Universal Robots PolyScope program: azat-test.urp

Program azat-test (installation=default directory=/programs createdIn=5.11.9.1010452 lastSavedIn=5.11.9.1010452 robotSerialNumber=20225200364)
Calibrated DH parameters: a=[0.00002, -0.569483, -0.54992, -0.00001, -0.000036, 0]; d=[0.180894, -146.691669, 192.918669, -46.053088, 0.119778, 0.115602]; alpha=[1.571425, -0.001534, 0.003359, 1.568739, -1.571477, 0]; deltaTheta=[0, 0.376258, -0.101074, -0.275185, -0.000002, 0]
Robot Program (runOnlyOnce=false)
  Script file /programs/usbdisk/Test.script
    | def Machining2():
    |   # Default parameters:
    |   global speed_ms = 0.3
    |   global speed_rads = 0.75
    |   global accel_mss = 3
    |   global accel_radss = 1.2
    |   global blend_radius_m = 0.001
    | 
    |   # Add subprograms here
    |   # Start of main program
    |   # Program generated by RoboDK v5.6.5 for UR10e on 11/10/2023 19:05:33
    |   # Using nominal kinematics.
    |   blend_radius_m = 0.001
    |   speed_ms = 1.000
    |   # set_reference(p[0.335000, -0.154000, 0.000000, 0.000000, 0.000000, 0.000000])
    |   set_tcp(p[0.000000, 0.000000, 0.252000, 0.000000, 0.000000, 0.000000])
    |   # Show Tool
    |   movej([0.093203, -1.219144, -2.564771, -0.928474, 1.570796, 1.664000],accel_radss,speed_rads,0,blend_radius_m)
    |   movel([0.093203, -1.219144, -2.564771, -0.928474, 1.570796, 1.664000],accel_mss,speed_ms,0,blend_radius_m)
    |   # Splitting Linear movement in 32 (instruction 7: MoveL 3)
    |   movel([0.093203, -1.220829, -2.565913, -0.925646, 1.570796, 1.664000],accel_mss,speed_ms,0,blend_radius_m)
    |   movel([0.093203, -1.222524, -2.567053, -0.922812, 1.570796, 1.664000],accel_mss,speed_ms,0,blend_radius_m)
    |   movel([0.093203, -1.224229, -2.568190, -0.919970, 1.570796, 1.664000],accel_mss,speed_ms,0,blend_radius_m)
    |   movel([0.093203, -1.225943, -2.569325, -0.917122, 1.570796, 1.664000],accel_mss,speed_ms,0,blend_radius_m)
    |   movel([0.093203, -1.227666, -2.570456, -0.914267, 1.570796, 1.664000],accel_mss,speed_ms,0,blend_radius_m)
    |   movel([0.093203, -1.229398, -2.571586, -0.911405, 1.570796, 1.664000],accel_mss,speed_ms,0,blend_radius_m)
    |   movel([0.093203, -1.231141, -2.572712, -0.908536, 1.570796, 1.664000],accel_mss,speed_ms,0,blend_radius_m)
    |   movel([0.093203, -1.232892, -2.573836, -0.905661, 1.570796, 1.664000],accel_mss,speed_ms,0,blend_radius_m)
    |   movel([0.093203, -1.234653, -2.574957, -0.902778, 1.570796, 1.664000],accel_mss,speed_ms,0,blend_radius_m)
    |   movel([0.093203, -1.236424, -2.576076, -0.899889, 1.570796, 1.664000],accel_mss,speed_ms,0,blend_radius_m)
    |   movel([0.093203, -1.238204, -2.577191, -0.896993, 1.570796, 1.664000],accel_mss,speed_ms,0,blend_radius_m)
    |   movel([0.093203, -1.239994, -2.578304, -0.894090, 1.570796, 1.664000],accel_mss,speed_ms,0,blend_radius_m)
    |   movel([0.093203, -1.241794, -2.579415, -0.891180, 1.570796, 1.664000],accel_mss,speed_ms,0,blend_radius_m)
    |   movel([0.093203, -1.243603, -2.580522, -0.888264, 1.570796, 1.664000],accel_mss,speed_ms,0,blend_radius_m)
    |   movel([0.093203, -1.245422, -2.581627, -0.885340, 1.570796, 1.664000],accel_mss,speed_ms,0,blend_radius_m)
    |   movel([0.093203, -1.247251, -2.582729, -0.882409, 1.570796, 1.664000],accel_mss,speed_ms,0,blend_radius_m)
    |   movel([0.093203, -1.249090, -2.583828, -0.879472, 1.570796, 1.664000],accel_mss,speed_ms,0,blend_radius_m)
    |   movel([0.093203, -1.250938, -2.584924, -0.876527, 1.570796, 1.664000],accel_mss,speed_ms,0,blend_radius_m)
    |   movel([0.093203, -1.252796, -2.586018, -0.873575, 1.570796, 1.664000],accel_mss,speed_ms,0,blend_radius_m)
    |   movel([0.093203, -1.254664, -2.587108, -0.870617, 1.570796, 1.664000],accel_mss,speed_ms,0,blend_radius_m)
    |   movel([0.093203, -1.256542, -2.588196, -0.867651, 1.570796, 1.664000],accel_mss,speed_ms,0,blend_radius_m)
    |   movel([0.093203, -1.258430, -2.589281, -0.864678, 1.570796, 1.664000],accel_mss,speed_ms,0,blend_radius_m)
    |   movel([0.093203, -1.260327, -2.590363, -0.861699, 1.570796, 1.664000],accel_mss,speed_ms,0,blend_radius_m)
    |   movel([0.093203, -1.262235, -2.591442, -0.858712, 1.570796, 1.664000],accel_mss,speed_ms,0,blend_radius_m)
    |   movel([0.093203, -1.264153, -2.592518, -0.855718, 1.570796, 1.664000],accel_mss,speed_ms,0,blend_radius_m)
    |   movel([0.093203, -1.266080, -2.593592, -0.852717, 1.570796, 1.664000],accel_mss,speed_ms,0,blend_radius_m)
    |   movel([0.093203, -1.268018, -2.594662, -0.849709, 1.570796, 1.664000],accel_mss,speed_ms,0,blend_radius_m)
    |   movel([0.093203, -1.269966, -2.595730, -0.846694, 1.570796, 1.664000],accel_mss,speed_ms,0,blend_radius_m)
    |   movel([0.093203, -1.271924, -2.596794, -0.843671, 1.570796, 1.664000],accel_mss,speed_ms,0,blend_radius_m)
    |   movel([0.093203, -1.273891, -2.597855, -0.840642, 1.570796, 1.664000],accel_mss,speed_ms,0,blend_radius_m)
    |   movel([0.093203, -1.275870, -2.598914, -0.837605, 1.570796, 1.664000],accel_mss,speed_ms,0,blend_radius_m)
    |   movel([0.093203, -1.277858, -2.599969, -0.834562, 1.570796, 1.664000],accel_mss,speed_ms,0,blend_radius_m)
    |   movel([0.093203, -1.277858, -2.599969, -0.834562, 1.570796, 1.664000],accel_mss,speed_ms,0,blend_radius_m)
    |   speed_ms = 1.000
    |   movel([0.093203, -1.277858, -2.599969, -0.834562, 1.570796, 1.664000],accel_mss,speed_ms,0,blend_radius_m)
    |   # Splitting Linear movement in 14 (instruction 11: MoveL 6)
    |   movel([0.093203, -1.279685, -2.600932, -0.831772, 1.570796, 1.664000],accel_mss,speed_ms,0,blend_radius_m)
    |   movel([0.093203, -1.281520, -2.601892, -0.828977, 1.570796, 1.664000],accel_mss,speed_ms,0,blend_radius_m)
    |   movel([0.093203, -1.283364, -2.602849, -0.826176, 1.570796, 1.664000],accel_mss,speed_ms,0,blend_radius_m)
    |   movel([0.093203, -1.285216, -2.603804, -0.823369, 1.570796, 1.664000],accel_mss,speed_ms,0,blend_radius_m)
    |   movel([0.093203, -1.287077, -2.604756, -0.820556, 1.570796, 1.664000],accel_mss,speed_ms,0,blend_radius_m)
    |   movel([0.093203, -1.288947, -2.605705, -0.817737, 1.570796, 1.664000],accel_mss,speed_ms,0,blend_radius_m)
    |   movel([0.093203, -1.290825, -2.606652, -0.814911, 1.570796, 1.664000],accel_mss,speed_ms,0,blend_radius_m)
    |   movel([0.093203, -1.292712, -2.607597, -0.812080, 1.570796, 1.664000],accel_mss,speed_ms,0,blend_radius_m)
    |   movel([0.093203, -1.294608, -2.608538, -0.809243, 1.570796, 1.664000],accel_mss,speed_ms,0,blend_radius_m)
    |   movel([0.093203, -1.296512, -2.609477, -0.806399, 1.570796, 1.664000],accel_mss,speed_ms,0,blend_radius_m)
    |   movel([0.093203, -1.298425, -2.610414, -0.803550, 1.570796, 1.664000],accel_mss,speed_ms,0,blend_radius_m)
    |   movel([0.093203, -1.300347, -2.611348, -0.800694, 1.570796, 1.664000],accel_mss,speed_ms,0,blend_radius_m)
    |   movel([0.093203, -1.302278, -2.612279, -0.797833, 1.570796, 1.664000],accel_mss,speed_ms,0,blend_radius_m)
    |   movel([0.093203, -1.304217, -2.613207, -0.794965, 1.570796, 1.664000],accel_mss,speed_ms,0,blend_radius_m)
    |   speed_ms = 0.003
    |   # Splitting Linear movement in 6 (instruction 13: MoveL 7)
    |   movel([0.093203, -1.305921, -2.614017, -0.792451, 1.570796, 1.664000],accel_mss,speed_ms,0,blend_radius_m)
    |   movel([0.093203, -1.307632, -2.614825, -0.789932, 1.570796, 1.664000],accel_mss,speed_ms,0,blend_radius_m)
    |   movel([0.093203, -1.309349, -2.615632, -0.787408, 1.570796, 1.664000],accel_mss,speed_ms,0,blend_radius_m)
    |   movel([0.093203, -1.311073, -2.616435, -0.784880, 1.570796, 1.664000],accel_mss,speed_ms,0,blend_radius_m)
    |   movel([0.093203, -1.312805, -2.617237, -0.782347, 1.570796, 1.664000],accel_mss,speed_ms,0,blend_radius_m)
    |   movel([0.093203, -1.314542, -2.618037, -0.779810, 1.570796, 1.664000],accel_mss,speed_ms,0,blend_radius_m)
    |   speed_ms = 0.007
    |   # Splitting Linear movement in 4 (instruction 15: MoveC 8)
    |   movel([0.093414, -1.312771, -2.619122, -0.780496, 1.570796, 1.664211],accel_mss,speed_ms,0,blend_radius_m)
    |   movel([0.093626, -1.310995, -2.620205, -0.781189, 1.570796, 1.664423],accel_mss,speed_ms,0,blend_radius_m)
    |   movel([0.093839, -1.309214, -2.621287, -0.781888, 1.570796, 1.664635],accel_mss,speed_ms,0,blend_radius_m)
    |   movel([0.094053, -1.307428, -2.622368, -0.782593, 1.570796, 1.664849],accel_mss,speed_ms,0,blend_radius_m)
    |   movel([0.094549, -1.306453, -2.622956, -0.782979, 1.570796, 1.665345],accel_mss,speed_ms,0,blend_radius_m)
    |   movel([0.095474, -1.305833, -2.623330, -0.783226, 1.570796, 1.666271],accel_mss,speed_ms,0,blend_radius_m)
    |   # Splitting Linear movement in 4 (instruction 18: MoveC 11)
    |   movel([0.097666, -1.305097, -2.623773, -0.783519, 1.570796, 1.668462],accel_mss,speed_ms,0,blend_radius_m)
    |   movel([0.099859, -1.304363, -2.624214, -0.783812, 1.570796, 1.670655],accel_mss,speed_ms,0,blend_radius_m)
    |   movel([0.102053, -1.303632, -2.624652, -0.784105, 1.570796, 1.672850],accel_mss,speed_ms,0,blend_radius_m)
    |   movel([0.104249, -1.302904, -2.625088, -0.784397, 1.570796, 1.675046],accel_mss,speed_ms,0,blend_radius_m)
    |   # Splitting Linear movement in 4 (instruction 19: MoveC 12)
    |   movel([0.106367, -1.302217, -2.625498, -0.784673, 1.570796, 1.677163],accel_mss,speed_ms,0,blend_radius_m)
    |   movel([0.108485, -1.301533, -2.625907, -0.784949, 1.570796, 1.679281],accel_mss,speed_ms,0,blend_radius_m)
    |   movel([0.110605, -1.300852, -2.626313, -0.785224, 1.570796, 1.681401],accel_mss,speed_ms,0,blend_radius_m)
    |   movel([0.112726, -1.300173, -2.626717, -0.785499, 1.570796, 1.683522],accel_mss,speed_ms,0,blend_radius_m)
    |   movel([0.114487, -1.299907, -2.626875, -0.785607, 1.570796, 1.685284],accel_mss,speed_ms,0,blend_radius_m)
    |   movel([0.114805, -1.300192, -2.626705, -0.785491, 1.570796, 1.685601],accel_mss,speed_ms,0,blend_radius_m)
    |   movel([0.114810, -1.301339, -2.626023, -0.785027, 1.570796, 1.685607],accel_mss,speed_ms,0,blend_radius_m)
    |   movel([0.114595, -1.303476, -2.624746, -0.784167, 1.570796, 1.685391],accel_mss,speed_ms,0,blend_radius_m)
    |   movel([0.113935, -1.308261, -2.621865, -0.782263, 1.570796, 1.684731],accel_mss,speed_ms,0,blend_radius_m)
    |   movel([0.113353, -1.312385, -2.619358, -0.780647, 1.570796, 1.684149],accel_mss,speed_ms,0,blend_radius_m)
    |   movel([0.112775, -1.316484, -2.616843, -0.779061, 1.570796, 1.683572],accel_mss,speed_ms,0,blend_radius_m)
    |   movel([0.107814, -1.318044, -2.615881, -0.778464, 1.570796, 1.678611],accel_mss,speed_ms,0,blend_radius_m)
    |   movel([0.102861, -1.319618, -2.614906, -0.777865, 1.570796, 1.673657],accel_mss,speed_ms,0,blend_radius_m)
    |   movel([0.097870, -1.321202, -2.613922, -0.777265, 1.570796, 1.668666],accel_mss,speed_ms,0,blend_radius_m)
    |   movel([0.094990, -1.322063, -2.613386, -0.776941, 1.570796, 1.665786],accel_mss,speed_ms,0,blend_radius_m)
    |   movel([0.093115, -1.322559, -2.613076, -0.776754, 1.570796, 1.663912],accel_mss,speed_ms,0,blend_radius_m)
    |   movel([0.092693, -1.322465, -2.613135, -0.776789, 1.570796, 1.663490],accel_mss,speed_ms,0,blend_radius_m)
    |   movel([0.092441, -1.321460, -2.613761, -0.777168, 1.570796, 1.663237],accel_mss,speed_ms,0,blend_radius_m)
    |   # Splitting Linear movement in 4 (instruction 34: MoveC 27)
    |   movel([0.092630, -1.319737, -2.614832, -0.777820, 1.570796, 1.663427],accel_mss,speed_ms,0,blend_radius_m)
    |   movel([0.092821, -1.318010, -2.615902, -0.778477, 1.570796, 1.663617],accel_mss,speed_ms,0,blend_radius_m)
    |   movel([0.093012, -1.316279, -2.616970, -0.779140, 1.570796, 1.663808],accel_mss,speed_ms,0,blend_radius_m)
    |   movel([0.093203, -1.314542, -2.618037, -0.779810, 1.570796, 1.664000],accel_mss,speed_ms,0,blend_radius_m)
    |   speed_ms = 0.003
    |   movel([0.093203, -1.318038, -2.619630, -0.774720, 1.570796, 1.664000],accel_mss,speed_ms,0,blend_radius_m)
    |   speed_ms = 0.007
    |   # Splitting Linear movement in 4 (instruction 38: MoveC 29)
    |   movel([0.093414, -1.316271, -2.620718, -0.775400, 1.570796, 1.664211],accel_mss,speed_ms,0,blend_radius_m)
    |   movel([0.093626, -1.314500, -2.621804, -0.776085, 1.570796, 1.664423],accel_mss,speed_ms,0,blend_radius_m)
    |   movel([0.093839, -1.312723, -2.622889, -0.776777, 1.570796, 1.664635],accel_mss,speed_ms,0,blend_radius_m)
    |   movel([0.094053, -1.310941, -2.623973, -0.777474, 1.570796, 1.664849],accel_mss,speed_ms,0,blend_radius_m)
    |   movel([0.094549, -1.309969, -2.624563, -0.777857, 1.570796, 1.665345],accel_mss,speed_ms,0,blend_radius_m)
    |   movel([0.095474, -1.309350, -2.624938, -0.778101, 1.570796, 1.666271],accel_mss,speed_ms,0,blend_radius_m)
    |   # Splitting Linear movement in 4 (instruction 41: MoveC 32)
    |   movel([0.097666, -1.308615, -2.625382, -0.778391, 1.570796, 1.668462],accel_mss,speed_ms,0,blend_radius_m)
    |   movel([0.099859, -1.307884, -2.625824, -0.778681, 1.570796, 1.670655],accel_mss,speed_ms,0,blend_radius_m)
    |   movel([0.102053, -1.307154, -2.626264, -0.778971, 1.570796, 1.672850],accel_mss,speed_ms,0,blend_radius_m)
    |   movel([0.104249, -1.306428, -2.626701, -0.779260, 1.570796, 1.675046],accel_mss,speed_ms,0,blend_radius_m)
    |   # Splitting Linear movement in 4 (instruction 42: MoveC 33)
    |   movel([0.106367, -1.305743, -2.627113, -0.779534, 1.570796, 1.677163],accel_mss,speed_ms,0,blend_radius_m)
    |   movel([0.108485, -1.305060, -2.627522, -0.779807, 1.570796, 1.679281],accel_mss,speed_ms,0,blend_radius_m)
    |   movel([0.110605, -1.304380, -2.627929, -0.780079, 1.570796, 1.681401],accel_mss,speed_ms,0,blend_radius_m)
    |   movel([0.112726, -1.303703, -2.628335, -0.780352, 1.570796, 1.683522],accel_mss,speed_ms,0,blend_radius_m)
    |   movel([0.114487, -1.303437, -2.628493, -0.780459, 1.570796, 1.685284],accel_mss,speed_ms,0,blend_radius_m)
    |   movel([0.114805, -1.303722, -2.628323, -0.780344, 1.570796, 1.685601],accel_mss,speed_ms,0,blend_radius_m)
    |   movel([0.114810, -1.304866, -2.627638, -0.779885, 1.570796, 1.685607],accel_mss,speed_ms,0,blend_radius_m)
    |   movel([0.114595, -1.306998, -2.626358, -0.779033, 1.570796, 1.685391],accel_mss,speed_ms,0,blend_radius_m)
    |   movel([0.113935, -1.311772, -2.623468, -0.777149, 1.570796, 1.684731],accel_mss,speed_ms,0,blend_radius_m)
    |   movel([0.113353, -1.315886, -2.620955, -0.775549, 1.570796, 1.684149],accel_mss,speed_ms,0,blend_radius_m)
    |   movel([0.112775, -1.319976, -2.618433, -0.773980, 1.570796, 1.683572],accel_mss,speed_ms,0,blend_radius_m)
    |   movel([0.107814, -1.321532, -2.617468, -0.773389, 1.570796, 1.678611],accel_mss,speed_ms,0,blend_radius_m)
    |   movel([0.102861, -1.323102, -2.616490, -0.772797, 1.570796, 1.673657],accel_mss,speed_ms,0,blend_radius_m)
    |   movel([0.097870, -1.324682, -2.615504, -0.772203, 1.570796, 1.668666],accel_mss,speed_ms,0,blend_radius_m)
    |   movel([0.094990, -1.325540, -2.614966, -0.771882, 1.570796, 1.665786],accel_mss,speed_ms,0,blend_radius_m)
    |   movel([0.093115, -1.326036, -2.614655, -0.771698, 1.570796, 1.663912],accel_mss,speed_ms,0,blend_radius_m)
    |   movel([0.092693, -1.325942, -2.614714, -0.771733, 1.570796, 1.663490],accel_mss,speed_ms,0,blend_radius_m)
    |   movel([0.092441, -1.324939, -2.615343, -0.772107, 1.570796, 1.663237],accel_mss,speed_ms,0,blend_radius_m)
    |   # Splitting Linear movement in 4 (instruction 57: MoveC 48)
    |   movel([0.092630, -1.323221, -2.616416, -0.772752, 1.570796, 1.663427],accel_mss,speed_ms,0,blend_radius_m)
    |   movel([0.092821, -1.321498, -2.617489, -0.773402, 1.570796, 1.663617],accel_mss,speed_ms,0,blend_radius_m)
    |   movel([0.093012, -1.319770, -2.618560, -0.774059, 1.570796, 1.663808],accel_mss,speed_ms,0,blend_radius_m)
    |   movel([0.093203, -1.318038, -2.619630, -0.774720, 1.570796, 1.664000],accel_mss,speed_ms,0,blend_radius_m)
    |   speed_ms = 0.003
    |   # Splitting Linear movement in 6 (instruction 59: MoveL 49)
    |   movel([0.093203, -1.315705, -2.618569, -0.778115, 1.570796, 1.664000],accel_mss,speed_ms,0,blend_radius_m)
    |   movel([0.093203, -1.313383, -2.617504, -0.781502, 1.570796, 1.664000],accel_mss,speed_ms,0,blend_radius_m)
    |   movel([0.093203, -1.311073, -2.616435, -0.784880, 1.570796, 1.664000],accel_mss,speed_ms,0,blend_radius_m)
    |   movel([0.093203, -1.308776, -2.615363, -0.788250, 1.570796, 1.664000],accel_mss,speed_ms,0,blend_radius_m)
    |   movel([0.093203, -1.306490, -2.614287, -0.791612, 1.570796, 1.664000],accel_mss,speed_ms,0,blend_radius_m)
    |   movel([0.093203, -1.304217, -2.613207, -0.794965, 1.570796, 1.664000],accel_mss,speed_ms,0,blend_radius_m)
    |   speed_ms = 1.000
    |   # Splitting Linear movement in 14 (instruction 61: MoveL 50)
    |   movel([0.093203, -1.302278, -2.612279, -0.797833, 1.570796, 1.664000],accel_mss,speed_ms,0,blend_radius_m)
    |   movel([0.093203, -1.300347, -2.611348, -0.800694, 1.570796, 1.664000],accel_mss,speed_ms,0,blend_radius_m)
    |   movel([0.093203, -1.298425, -2.610414, -0.803550, 1.570796, 1.664000],accel_mss,speed_ms,0,blend_radius_m)
    |   movel([0.093203, -1.296512, -2.609477, -0.806399, 1.570796, 1.664000],accel_mss,speed_ms,0,blend_radius_m)
    |   movel([0.093203, -1.294608, -2.608538, -0.809243, 1.570796, 1.664000],accel_mss,speed_ms,0,blend_radius_m)
    |   movel([0.093203, -1.292712, -2.607597, -0.812080, 1.570796, 1.664000],accel_mss,speed_ms,0,blend_radius_m)
    |   movel([0.093203, -1.290825, -2.606652, -0.814911, 1.570796, 1.664000],accel_mss,speed_ms,0,blend_radius_m)
    |   movel([0.093203, -1.288947, -2.605705, -0.817737, 1.570796, 1.664000],accel_mss,speed_ms,0,blend_radius_m)
    |   movel([0.093203, -1.287077, -2.604756, -0.820556, 1.570796, 1.664000],accel_mss,speed_ms,0,blend_radius_m)
    |   movel([0.093203, -1.285216, -2.603804, -0.823369, 1.570796, 1.664000],accel_mss,speed_ms,0,blend_radius_m)
    |   movel([0.093203, -1.283364, -2.602849, -0.826176, 1.570796, 1.664000],accel_mss,speed_ms,0,blend_radius_m)
    |   movel([0.093203, -1.281520, -2.601892, -0.828977, 1.570796, 1.664000],accel_mss,speed_ms,0,blend_radius_m)
    |   movel([0.093203, -1.279685, -2.600932, -0.831772, 1.570796, 1.664000],accel_mss,speed_ms,0,blend_radius_m)
    |   movel([0.093203, -1.277858, -2.599969, -0.834562, 1.570796, 1.664000],accel_mss,speed_ms,0,blend_radius_m)
    |   movel([0.096025, -1.277288, -2.600301, -0.834800, 1.570796, 1.666821],accel_mss,speed_ms,0,blend_radius_m)
    |   # Splitting Linear movement in 14 (instruction 63: MoveL 52)
    |   movel([0.096025, -1.279116, -2.601264, -0.832010, 1.570796, 1.666821],accel_mss,speed_ms,0,blend_radius_m)
    |   movel([0.096025, -1.280952, -2.602224, -0.829213, 1.570796, 1.666821],accel_mss,speed_ms,0,blend_radius_m)
    |   movel([0.096025, -1.282796, -2.603182, -0.826411, 1.570796, 1.666821],accel_mss,speed_ms,0,blend_radius_m)
    |   movel([0.096025, -1.284649, -2.604137, -0.823603, 1.570796, 1.666821],accel_mss,speed_ms,0,blend_radius_m)
    |   movel([0.096025, -1.286511, -2.605090, -0.820789, 1.570796, 1.666821],accel_mss,speed_ms,0,blend_radius_m)
    |   movel([0.096025, -1.288381, -2.606040, -0.817968, 1.570796, 1.666821],accel_mss,speed_ms,0,blend_radius_m)
    |   movel([0.096025, -1.290260, -2.606987, -0.815142, 1.570796, 1.666821],accel_mss,speed_ms,0,blend_radius_m)
    |   movel([0.096025, -1.292147, -2.607932, -0.812309, 1.570796, 1.666821],accel_mss,speed_ms,0,blend_radius_m)
    |   movel([0.096025, -1.294044, -2.608874, -0.809471, 1.570796, 1.666821],accel_mss,speed_ms,0,blend_radius_m)
    |   movel([0.096025, -1.295949, -2.609814, -0.806626, 1.570796, 1.666821],accel_mss,speed_ms,0,blend_radius_m)
    |   movel([0.096025, -1.297862, -2.610751, -0.803776, 1.570796, 1.666821],accel_mss,speed_ms,0,blend_radius_m)
    |   movel([0.096025, -1.299785, -2.611685, -0.800919, 1.570796, 1.666821],accel_mss,speed_ms,0,blend_radius_m)
    |   movel([0.096025, -1.301716, -2.612617, -0.798056, 1.570796, 1.666821],accel_mss,speed_ms,0,blend_radius_m)
    |   movel([0.096025, -1.303656, -2.613546, -0.795187, 1.570796, 1.666821],accel_mss,speed_ms,0,blend_radius_m)
    |   speed_ms = 0.003
    |   # Splitting Linear movement in 6 (instruction 65: MoveL 53)
    |   movel([0.096025, -1.305361, -2.614357, -0.792672, 1.570796, 1.666821],accel_mss,speed_ms,0,blend_radius_m)
    |   movel([0.096025, -1.307072, -2.615165, -0.790152, 1.570796, 1.666821],accel_mss,speed_ms,0,blend_radius_m)
    |   movel([0.096025, -1.308790, -2.615972, -0.787627, 1.570796, 1.666821],accel_mss,speed_ms,0,blend_radius_m)
    |   movel([0.096025, -1.310515, -2.616776, -0.785098, 1.570796, 1.666821],accel_mss,speed_ms,0,blend_radius_m)
    |   movel([0.096025, -1.312247, -2.617579, -0.782564, 1.570796, 1.666821],accel_mss,speed_ms,0,blend_radius_m)
    |   movel([0.096025, -1.313985, -2.618379, -0.780025, 1.570796, 1.666821],accel_mss,speed_ms,0,blend_radius_m)
    |   speed_ms = 0.007
    |   movel([0.096371, -1.312310, -2.619403, -0.780676, 1.570796, 1.667168],accel_mss,speed_ms,0,blend_radius_m)
    |   movel([0.097026, -1.310764, -2.620346, -0.781279, 1.570796, 1.667822],accel_mss,speed_ms,0,blend_radius_m)
    |   movel([0.097647, -1.310126, -2.620733, -0.781529, 1.570796, 1.668443],accel_mss,speed_ms,0,blend_radius_m)
    |   movel([0.098109, -1.310180, -2.620701, -0.781508, 1.570796, 1.668906],accel_mss,speed_ms,0,blend_radius_m)
    |   movel([0.098200, -1.310314, -2.620619, -0.781456, 1.570796, 1.668996],accel_mss,speed_ms,0,blend_radius_m)
    |   movel([0.098382, -1.310404, -2.620564, -0.781420, 1.570796, 1.669178],accel_mss,speed_ms,0,blend_radius_m)
    |   movel([0.098620, -1.310445, -2.620540, -0.781404, 1.570796, 1.669416],accel_mss,speed_ms,0,blend_radius_m)
    |   movel([0.098880, -1.310424, -2.620552, -0.781412, 1.570796, 1.669676],accel_mss,speed_ms,0,blend_radius_m)
    |   movel([0.099778, -1.310438, -2.620544, -0.781407, 1.570796, 1.670575],accel_mss,speed_ms,0,blend_radius_m)
    |   movel([0.100980, -1.310873, -2.620279, -0.781237, 1.570796, 1.671777],accel_mss,speed_ms,0,blend_radius_m)
    |   movel([0.102074, -1.311483, -2.619908, -0.780998, 1.570796, 1.672870],accel_mss,speed_ms,0,blend_radius_m)
    |   movel([0.102637, -1.312124, -2.619517, -0.780748, 1.570796, 1.673434],accel_mss,speed_ms,0,blend_radius_m)
    |   movel([0.103095, -1.312584, -2.619236, -0.780569, 1.570796, 1.673891],accel_mss,speed_ms,0,blend_radius_m)
    |   movel([0.103752, -1.312653, -2.619194, -0.780542, 1.570796, 1.674549],accel_mss,speed_ms,0,blend_radius_m)
    |   movel([0.104468, -1.312318, -2.619398, -0.780673, 1.570796, 1.675265],accel_mss,speed_ms,0,blend_radius_m)
    |   movel([0.105100, -1.311655, -2.619803, -0.780931, 1.570796, 1.675897],accel_mss,speed_ms,0,blend_radius_m)
    |   movel([0.105382, -1.310966, -2.620223, -0.781200, 1.570796, 1.676178],accel_mss,speed_ms,0,blend_radius_m)
    |   movel([0.105257, -1.310406, -2.620564, -0.781420, 1.570796, 1.676054],accel_mss,speed_ms,0,blend_radius_m)
    |   movel([0.104714, -1.310070, -2.620768, -0.781551, 1.570796, 1.675511],accel_mss,speed_ms,0,blend_radius_m)
    |   movel([0.103830, -1.310013, -2.620802, -0.781574, 1.570796, 1.674626],accel_mss,speed_ms,0,blend_radius_m)
    |   movel([0.102821, -1.309943, -2.620845, -0.781601, 1.570796, 1.673617],accel_mss,speed_ms,0,blend_radius_m)
    |   movel([0.101620, -1.309547, -2.621085, -0.781757, 1.570796, 1.672416],accel_mss,speed_ms,0,blend_radius_m)
    |   movel([0.100579, -1.309026, -2.621401, -0.781962, 1.570796, 1.671375],accel_mss,speed_ms,0,blend_radius_m)
    |   movel([0.100378, -1.308566, -2.621680, -0.782143, 1.570796, 1.671175],accel_mss,speed_ms,0,blend_radius_m)
    |   movel([0.100338, -1.308416, -2.621771, -0.782202, 1.570796, 1.671134],accel_mss,speed_ms,0,blend_radius_m)
    |   movel([0.100177, -1.308298, -2.621842, -0.782249, 1.570796, 1.670973],accel_mss,speed_ms,0,blend_radius_m)
    |   movel([0.099929, -1.308228, -2.621885, -0.782276, 1.570796, 1.670725],accel_mss,speed_ms,0,blend_radius_m)
    |   movel([0.099627, -1.308219, -2.621890, -0.782280, 1.570796, 1.670423],accel_mss,speed_ms,0,blend_radius_m)
    |   movel([0.099329, -1.308173, -2.621918, -0.782298, 1.570796, 1.670125],accel_mss,speed_ms,0,blend_radius_m)
    |   movel([0.099332, -1.308004, -2.622020, -0.782365, 1.570796, 1.670128],accel_mss,speed_ms,0,blend_radius_m)
    |   movel([0.099696, -1.307652, -2.622233, -0.782504, 1.570796, 1.670493],accel_mss,speed_ms,0,blend_radius_m)
    |   movel([0.100739, -1.306867, -2.622707, -0.782815, 1.570796, 1.671535],accel_mss,speed_ms,0,blend_radius_m)
    |   movel([0.101828, -1.306120, -2.623157, -0.783112, 1.570796, 1.672625],accel_mss,speed_ms,0,blend_radius_m)
    |   movel([0.102774, -1.305602, -2.623469, -0.783318, 1.570796, 1.673570],accel_mss,speed_ms,0,blend_radius_m)
    |   movel([0.103807, -1.305194, -2.623715, -0.783480, 1.570796, 1.674604],accel_mss,speed_ms,0,blend_radius_m)
    |   movel([0.105195, -1.304789, -2.623958, -0.783642, 1.570796, 1.675992],accel_mss,speed_ms,0,blend_radius_m)
    |   movel([0.107386, -1.304416, -2.624182, -0.783791, 1.570796, 1.678182],accel_mss,speed_ms,0,blend_radius_m)
    |   movel([0.109163, -1.304547, -2.624103, -0.783739, 1.570796, 1.679959],accel_mss,speed_ms,0,blend_radius_m)
    |   movel([0.110515, -1.305193, -2.623716, -0.783481, 1.570796, 1.681312],accel_mss,speed_ms,0,blend_radius_m)
    |   movel([0.111455, -1.306330, -2.623031, -0.783028, 1.570796, 1.682252],accel_mss,speed_ms,0,blend_radius_m)
    |   movel([0.111894, -1.307521, -2.622312, -0.782556, 1.570796, 1.682691],accel_mss,speed_ms,0,blend_radius_m)
    |   movel([0.111953, -1.308692, -2.621604, -0.782094, 1.570796, 1.682750],accel_mss,speed_ms,0,blend_radius_m)
    |   movel([0.111624, -1.309990, -2.620817, -0.781583, 1.570796, 1.682420],accel_mss,speed_ms,0,blend_radius_m)
    |   movel([0.110890, -1.311551, -2.619866, -0.780972, 1.570796, 1.681687],accel_mss,speed_ms,0,blend_radius_m)
    |   movel([0.109871, -1.313067, -2.618940, -0.780381, 1.570796, 1.680668],accel_mss,speed_ms,0,blend_radius_m)
    |   movel([0.108527, -1.314515, -2.618054, -0.779820, 1.570796, 1.679323],accel_mss,speed_ms,0,blend_radius_m)
    |   movel([0.106940, -1.315814, -2.617256, -0.779319, 1.570796, 1.677737],accel_mss,speed_ms,0,blend_radius_m)
    |   movel([0.105199, -1.316892, -2.616592, -0.778905, 1.570796, 1.675995],accel_mss,speed_ms,0,blend_radius_m)
    |   movel([0.101733, -1.318082, -2.615857, -0.778450, 1.570796, 1.672529],accel_mss,speed_ms,0,blend_radius_m)
    |   movel([0.098619, -1.317912, -2.615962, -0.778515, 1.570796, 1.669416],accel_mss,speed_ms,0,blend_radius_m)
    |   movel([0.096557, -1.316443, -2.616869, -0.779077, 1.570796, 1.667353],accel_mss,speed_ms,0,blend_radius_m)
    |   movel([0.096025, -1.313985, -2.618379, -0.780025, 1.570796, 1.666821],accel_mss,speed_ms,0,blend_radius_m)
    |   speed_ms = 0.003
    |   movel([0.096025, -1.317482, -2.619973, -0.774934, 1.570796, 1.666821],accel_mss,speed_ms,0,blend_radius_m)
    |   speed_ms = 0.007
    |   movel([0.096371, -1.315811, -2.621000, -0.775577, 1.570796, 1.667168],accel_mss,speed_ms,0,blend_radius_m)
    |   movel([0.097026, -1.314269, -2.621945, -0.776175, 1.570796, 1.667822],accel_mss,speed_ms,0,blend_radius_m)
    |   movel([0.097647, -1.313633, -2.622334, -0.776422, 1.570796, 1.668443],accel_mss,speed_ms,0,blend_radius_m)
    |   movel([0.098109, -1.313687, -2.622301, -0.776401, 1.570796, 1.668906],accel_mss,speed_ms,0,blend_radius_m)
    |   movel([0.098200, -1.313820, -2.622220, -0.776349, 1.570796, 1.668996],accel_mss,speed_ms,0,blend_radius_m)
    |   movel([0.098382, -1.313910, -2.622165, -0.776314, 1.570796, 1.669178],accel_mss,speed_ms,0,blend_radius_m)
    |   movel([0.098620, -1.313950, -2.622140, -0.776299, 1.570796, 1.669416],accel_mss,speed_ms,0,blend_radius_m)
    |   movel([0.098880, -1.313930, -2.622152, -0.776306, 1.570796, 1.669676],accel_mss,speed_ms,0,blend_radius_m)
    |   movel([0.099778, -1.313944, -2.622144, -0.776301, 1.570796, 1.670575],accel_mss,speed_ms,0,blend_radius_m)
    |   movel([0.100980, -1.314378, -2.621879, -0.776132, 1.570796, 1.671777],accel_mss,speed_ms,0,blend_radius_m)
    |   movel([0.102074, -1.314986, -2.621506, -0.775897, 1.570796, 1.672870],accel_mss,speed_ms,0,blend_radius_m)
    |   movel([0.102637, -1.315625, -2.621114, -0.775649, 1.570796, 1.673434],accel_mss,speed_ms,0,blend_radius_m)
    |   movel([0.103095, -1.316085, -2.620832, -0.775472, 1.570796, 1.673891],accel_mss,speed_ms,0,blend_radius_m)
    |   movel([0.103752, -1.316154, -2.620790, -0.775445, 1.570796, 1.674549],accel_mss,speed_ms,0,blend_radius_m)
    |   movel([0.104468, -1.315819, -2.620995, -0.775574, 1.570796, 1.675265],accel_mss,speed_ms,0,blend_radius_m)
    |   movel([0.105100, -1.315157, -2.621401, -0.775830, 1.570796, 1.675897],accel_mss,speed_ms,0,blend_radius_m)
    |   movel([0.105382, -1.314470, -2.621822, -0.776097, 1.570796, 1.676178],accel_mss,speed_ms,0,blend_radius_m)
    |   movel([0.105257, -1.313912, -2.622164, -0.776314, 1.570796, 1.676054],accel_mss,speed_ms,0,blend_radius_m)
    |   movel([0.104714, -1.313576, -2.622369, -0.776444, 1.570796, 1.675511],accel_mss,speed_ms,0,blend_radius_m)
    |   movel([0.103830, -1.313520, -2.622403, -0.776466, 1.570796, 1.674626],accel_mss,speed_ms,0,blend_radius_m)
    |   movel([0.102821, -1.313450, -2.622446, -0.776493, 1.570796, 1.673617],accel_mss,speed_ms,0,blend_radius_m)
    |   movel([0.101620, -1.313055, -2.622687, -0.776647, 1.570796, 1.672416],accel_mss,speed_ms,0,blend_radius_m)
    |   movel([0.100579, -1.312535, -2.623004, -0.776850, 1.570796, 1.671375],accel_mss,speed_ms,0,blend_radius_m)
    |   movel([0.100378, -1.312077, -2.623283, -0.777029, 1.570796, 1.671175],accel_mss,speed_ms,0,blend_radius_m)
    |   movel([0.100338, -1.311927, -2.623374, -0.777088, 1.570796, 1.671134],accel_mss,speed_ms,0,blend_radius_m)
    |   movel([0.100177, -1.311809, -2.623446, -0.777134, 1.570796, 1.670973],accel_mss,speed_ms,0,blend_radius_m)
    |   movel([0.099929, -1.311739, -2.623489, -0.777162, 1.570796, 1.670725],accel_mss,speed_ms,0,blend_radius_m)
    |   movel([0.099627, -1.311730, -2.623494, -0.777165, 1.570796, 1.670423],accel_mss,speed_ms,0,blend_radius_m)
    |   movel([0.099329, -1.311684, -2.623522, -0.777183, 1.570796, 1.670125],accel_mss,speed_ms,0,blend_radius_m)
    |   movel([0.099332, -1.311515, -2.623624, -0.777249, 1.570796, 1.670128],accel_mss,speed_ms,0,blend_radius_m)
    |   movel([0.099696, -1.311164, -2.623838, -0.777387, 1.570796, 1.670493],accel_mss,speed_ms,0,blend_radius_m)
    |   movel([0.100739, -1.310381, -2.624313, -0.777695, 1.570796, 1.671535],accel_mss,speed_ms,0,blend_radius_m)
    |   movel([0.101828, -1.309636, -2.624765, -0.777988, 1.570796, 1.672625],accel_mss,speed_ms,0,blend_radius_m)
    |   movel([0.102774, -1.309119, -2.625078, -0.778192, 1.570796, 1.673570],accel_mss,speed_ms,0,blend_radius_m)
    |   movel([0.103807, -1.308712, -2.625324, -0.778353, 1.570796, 1.674604],accel_mss,speed_ms,0,blend_radius_m)
    |   movel([0.105195, -1.308308, -2.625568, -0.778513, 1.570796, 1.675992],accel_mss,speed_ms,0,blend_radius_m)
    |   movel([0.107386, -1.307936, -2.625792, -0.778661, 1.570796, 1.678182],accel_mss,speed_ms,0,blend_radius_m)
    |   movel([0.109163, -1.308067, -2.625714, -0.778609, 1.570796, 1.679959],accel_mss,speed_ms,0,blend_radius_m)
    |   movel([0.110515, -1.308711, -2.625325, -0.778354, 1.570796, 1.681312],accel_mss,speed_ms,0,blend_radius_m)
    |   movel([0.111455, -1.309845, -2.624638, -0.777906, 1.570796, 1.682252],accel_mss,speed_ms,0,blend_radius_m)
    |   movel([0.111894, -1.311033, -2.623918, -0.777438, 1.570796, 1.682691],accel_mss,speed_ms,0,blend_radius_m)
    |   movel([0.111953, -1.312201, -2.623207, -0.776980, 1.570796, 1.682750],accel_mss,speed_ms,0,blend_radius_m)
    |   movel([0.111624, -1.313496, -2.622417, -0.776475, 1.570796, 1.682420],accel_mss,speed_ms,0,blend_radius_m)
    |   movel([0.110890, -1.315054, -2.621465, -0.775870, 1.570796, 1.681687],accel_mss,speed_ms,0,blend_radius_m)
    |   movel([0.109871, -1.316567, -2.620536, -0.775286, 1.570796, 1.680668],accel_mss,speed_ms,0,blend_radius_m)
    |   movel([0.108527, -1.318011, -2.619647, -0.774731, 1.570796, 1.679323],accel_mss,speed_ms,0,blend_radius_m)
    |   movel([0.106940, -1.319307, -2.618847, -0.774235, 1.570796, 1.677737],accel_mss,speed_ms,0,blend_radius_m)
    |   movel([0.105199, -1.320382, -2.618181, -0.773826, 1.570796, 1.675995],accel_mss,speed_ms,0,blend_radius_m)
    |   movel([0.101733, -1.321569, -2.617444, -0.773375, 1.570796, 1.672529],accel_mss,speed_ms,0,blend_radius_m)
    |   movel([0.098619, -1.321400, -2.617550, -0.773440, 1.570796, 1.669416],accel_mss,speed_ms,0,blend_radius_m)
    |   movel([0.096557, -1.319934, -2.618459, -0.773996, 1.570796, 1.667353],accel_mss,speed_ms,0,blend_radius_m)
    |   movel([0.096025, -1.317482, -2.619973, -0.774934, 1.570796, 1.666821],accel_mss,speed_ms,0,blend_radius_m)
    |   speed_ms = 0.003
    |   # Splitting Linear movement in 6 (instruction 175: MoveL 159)
    |   movel([0.096025, -1.315148, -2.618911, -0.778330, 1.570796, 1.666821],accel_mss,speed_ms,0,blend_radius_m)
    |   movel([0.096025, -1.312825, -2.617845, -0.781718, 1.570796, 1.666821],accel_mss,speed_ms,0,blend_radius_m)
    |   movel([0.096025, -1.310515, -2.616776, -0.785098, 1.570796, 1.666821],accel_mss,speed_ms,0,blend_radius_m)
    |   movel([0.096025, -1.308217, -2.615703, -0.788469, 1.570796, 1.666821],accel_mss,speed_ms,0,blend_radius_m)
    |   movel([0.096025, -1.305930, -2.614626, -0.791832, 1.570796, 1.666821],accel_mss,speed_ms,0,blend_radius_m)
    |   movel([0.096025, -1.303656, -2.613546, -0.795187, 1.570796, 1.666821],accel_mss,speed_ms,0,blend_radius_m)
    |   speed_ms = 1.000
    |   # Splitting Linear movement in 14 (instruction 177: MoveL 160)
    |   movel([0.096025, -1.301716, -2.612617, -0.798056, 1.570796, 1.666821],accel_mss,speed_ms,0,blend_radius_m)
    |   movel([0.096025, -1.299785, -2.611685, -0.800919, 1.570796, 1.666821],accel_mss,speed_ms,0,blend_radius_m)
    |   movel([0.096025, -1.297862, -2.610751, -0.803776, 1.570796, 1.666821],accel_mss,speed_ms,0,blend_radius_m)
    |   movel([0.096025, -1.295949, -2.609814, -0.806626, 1.570796, 1.666821],accel_mss,speed_ms,0,blend_radius_m)
    |   movel([0.096025, -1.294044, -2.608874, -0.809471, 1.570796, 1.666821],accel_mss,speed_ms,0,blend_radius_m)
    |   movel([0.096025, -1.292147, -2.607932, -0.812309, 1.570796, 1.666821],accel_mss,speed_ms,0,blend_radius_m)
    |   movel([0.096025, -1.290260, -2.606987, -0.815142, 1.570796, 1.666821],accel_mss,speed_ms,0,blend_radius_m)
    |   movel([0.096025, -1.288381, -2.606040, -0.817968, 1.570796, 1.666821],accel_mss,speed_ms,0,blend_radius_m)
    |   movel([0.096025, -1.286511, -2.605090, -0.820789, 1.570796, 1.666821],accel_mss,speed_ms,0,blend_radius_m)
    |   movel([0.096025, -1.284649, -2.604137, -0.823603, 1.570796, 1.666821],accel_mss,speed_ms,0,blend_radius_m)
    |   movel([0.096025, -1.282796, -2.603182, -0.826411, 1.570796, 1.666821],accel_mss,speed_ms,0,blend_radius_m)
    |   movel([0.096025, -1.280952, -2.602224, -0.829213, 1.570796, 1.666821],accel_mss,speed_ms,0,blend_radius_m)
    |   movel([0.096025, -1.279116, -2.601264, -0.832010, 1.570796, 1.666821],accel_mss,speed_ms,0,blend_radius_m)
    |   movel([0.096025, -1.277288, -2.600301, -0.834800, 1.570796, 1.666821],accel_mss,speed_ms,0,blend_radius_m)
    |   # Splitting Linear movement in 6 (instruction 178: MoveL 161)
    |   movel([0.096617, -1.278984, -2.599313, -0.834092, 1.570796, 1.667413],accel_mss,speed_ms,0,blend_radius_m)
    |   movel([0.097207, -1.280676, -2.598324, -0.833389, 1.570796, 1.668003],accel_mss,speed_ms,0,blend_radius_m)
    |   movel([0.097795, -1.282366, -2.597333, -0.832690, 1.570796, 1.668591],accel_mss,speed_ms,0,blend_radius_m)
    |   movel([0.098379, -1.284053, -2.596339, -0.831996, 1.570796, 1.669176],accel_mss,speed_ms,0,blend_radius_m)
    |   movel([0.098962, -1.285738, -2.595344, -0.831307, 1.570796, 1.669758],accel_mss,speed_ms,0,blend_radius_m)
    |   movel([0.099542, -1.287421, -2.594346, -0.830622, 1.570796, 1.670338],accel_mss,speed_ms,0,blend_radius_m)
    |   # Splitting Linear movement in 12 (instruction 179: MoveL 162)
    |   movel([0.099542, -1.289542, -2.595458, -0.827389, 1.570796, 1.670338],accel_mss,speed_ms,0,blend_radius_m)
    |   movel([0.099542, -1.291675, -2.596567, -0.824147, 1.570796, 1.670338],accel_mss,speed_ms,0,blend_radius_m)
    |   movel([0.099542, -1.293819, -2.597672, -0.820898, 1.570796, 1.670338],accel_mss,speed_ms,0,blend_radius_m)
    |   movel([0.099542, -1.295975, -2.598774, -0.817641, 1.570796, 1.670338],accel_mss,speed_ms,0,blend_radius_m)
    |   movel([0.099542, -1.298142, -2.599872, -0.814375, 1.570796, 1.670338],accel_mss,speed_ms,0,blend_radius_m)
    |   movel([0.099542, -1.300321, -2.600966, -0.811102, 1.570796, 1.670338],accel_mss,speed_ms,0,blend_radius_m)
    |   movel([0.099542, -1.302511, -2.602057, -0.807821, 1.570796, 1.670338],accel_mss,speed_ms,0,blend_radius_m)
    |   movel([0.099542, -1.304712, -2.603145, -0.804532, 1.570796, 1.670338],accel_mss,speed_ms,0,blend_radius_m)
    |   movel([0.099542, -1.306925, -2.604228, -0.801235, 1.570796, 1.670338],accel_mss,speed_ms,0,blend_radius_m)
    |   movel([0.099542, -1.309150, -2.605309, -0.797930, 1.570796, 1.670338],accel_mss,speed_ms,0,blend_radius_m)
    |   movel([0.099542, -1.311387, -2.606385, -0.794617, 1.570796, 1.670338],accel_mss,speed_ms,0,blend_radius_m)
    |   movel([0.099542, -1.313635, -2.607458, -0.791296, 1.570796, 1.670338],accel_mss,speed_ms,0,blend_radius_m)
    |   speed_ms = 0.003
    |   # Splitting Linear movement in 6 (instruction 181: MoveL 163)
    |   movel([0.099542, -1.315328, -2.608260, -0.788800, 1.570796, 1.670338],accel_mss,speed_ms,0,blend_radius_m)
    |   movel([0.099542, -1.317029, -2.609061, -0.786300, 1.570796, 1.670338],accel_mss,speed_ms,0,blend_radius_m)
    |   movel([0.099542, -1.318736, -2.609859, -0.783795, 1.570796, 1.670338],accel_mss,speed_ms,0,blend_radius_m)
    |   movel([0.099542, -1.320449, -2.610655, -0.781285, 1.570796, 1.670338],accel_mss,speed_ms,0,blend_radius_m)
    |   movel([0.099542, -1.322169, -2.611449, -0.778771, 1.570796, 1.670338],accel_mss,speed_ms,0,blend_radius_m)
    |   movel([0.099542, -1.323896, -2.612241, -0.776253, 1.570796, 1.670338],accel_mss,speed_ms,0,blend_radius_m)
    |   speed_ms = 0.007
    |   movel([0.099826, -1.323723, -2.612349, -0.776317, 1.570796, 1.670622],accel_mss,speed_ms,0,blend_radius_m)
    |   movel([0.100093, -1.323725, -2.612348, -0.776317, 1.570796, 1.670889],accel_mss,speed_ms,0,blend_radius_m)
    |   movel([0.100254, -1.323902, -2.612236, -0.776250, 1.570796, 1.671050],accel_mss,speed_ms,0,blend_radius_m)
    |   movel([0.100313, -1.324291, -2.611993, -0.776105, 1.570796, 1.671109],accel_mss,speed_ms,0,blend_radius_m)
    |   movel([0.100269, -1.324944, -2.611584, -0.775861, 1.570796, 1.671066],accel_mss,speed_ms,0,blend_radius_m)
    |   movel([0.100218, -1.325709, -2.611103, -0.775576, 1.570796, 1.671014],accel_mss,speed_ms,0,blend_radius_m)
    |   movel([0.100312, -1.326084, -2.610867, -0.775437, 1.570796, 1.671108],accel_mss,speed_ms,0,blend_radius_m)
    |   movel([0.100577, -1.326247, -2.610765, -0.775377, 1.570796, 1.671374],accel_mss,speed_ms,0,blend_radius_m)
    |   movel([0.101087, -1.326263, -2.610755, -0.775371, 1.570796, 1.671883],accel_mss,speed_ms,0,blend_radius_m)
    |   movel([0.101527, -1.326279, -2.610745, -0.775365, 1.570796, 1.672323],accel_mss,speed_ms,0,blend_radius_m)
    |   movel([0.102040, -1.326417, -2.610658, -0.775314, 1.570796, 1.672837],accel_mss,speed_ms,0,blend_radius_m)
    |   movel([0.102538, -1.326638, -2.610519, -0.775232, 1.570796, 1.673335],accel_mss,speed_ms,0,blend_radius_m)
    |   movel([0.102947, -1.326914, -2.610345, -0.775130, 1.570796, 1.673743],accel_mss,speed_ms,0,blend_radius_m)
    |   movel([0.103665, -1.328146, -2.609568, -0.774675, 1.570796, 1.674461],accel_mss,speed_ms,0,blend_radius_m)
    |   movel([0.103516, -1.329776, -2.608536, -0.774076, 1.570796, 1.674312],accel_mss,speed_ms,0,blend_radius_m)
    |   movel([0.102517, -1.331523, -2.607427, -0.773439, 1.570796, 1.673313],accel_mss,speed_ms,0,blend_radius_m)
    |   movel([0.100855, -1.333086, -2.606431, -0.772872, 1.570796, 1.671651],accel_mss,speed_ms,0,blend_radius_m)
    |   movel([0.100194, -1.333615, -2.606093, -0.772681, 1.570796, 1.670991],accel_mss,speed_ms,0,blend_radius_m)
    |   movel([0.099818, -1.334062, -2.605807, -0.772520, 1.570796, 1.670614],accel_mss,speed_ms,0,blend_radius_m)
    |   movel([0.099600, -1.334579, -2.605476, -0.772334, 1.570796, 1.670396],accel_mss,speed_ms,0,blend_radius_m)
    |   movel([0.099465, -1.335357, -2.604978, -0.772054, 1.570796, 1.670261],accel_mss,speed_ms,0,blend_radius_m)
    |   movel([0.099351, -1.336107, -2.604496, -0.771786, 1.570796, 1.670148],accel_mss,speed_ms,0,blend_radius_m)
    |   movel([0.099189, -1.336523, -2.604229, -0.771637, 1.570796, 1.669985],accel_mss,speed_ms,0,blend_radius_m)
    |   movel([0.098926, -1.336788, -2.604058, -0.771543, 1.570796, 1.669723],accel_mss,speed_ms,0,blend_radius_m)
    |   movel([0.098514, -1.336979, -2.603936, -0.771475, 1.570796, 1.669311],accel_mss,speed_ms,0,blend_radius_m)
    |   movel([0.098117, -1.337033, -2.603901, -0.771456, 1.570796, 1.668914],accel_mss,speed_ms,0,blend_radius_m)
    |   movel([0.097898, -1.336914, -2.603977, -0.771498, 1.570796, 1.668695],accel_mss,speed_ms,0,blend_radius_m)
    |   movel([0.097822, -1.336566, -2.604201, -0.771622, 1.570796, 1.668619],accel_mss,speed_ms,0,blend_radius_m)
    |   movel([0.097878, -1.335823, -2.604679, -0.771887, 1.570796, 1.668674],accel_mss,speed_ms,0,blend_radius_m)
    |   movel([0.097922, -1.335089, -2.605150, -0.772151, 1.570796, 1.668718],accel_mss,speed_ms,0,blend_radius_m)
    |   movel([0.097831, -1.334687, -2.605407, -0.772295, 1.570796, 1.668627],accel_mss,speed_ms,0,blend_radius_m)
    |   movel([0.097583, -1.334478, -2.605541, -0.772370, 1.570796, 1.668379],accel_mss,speed_ms,0,blend_radius_m)
    |   movel([0.097128, -1.334398, -2.605592, -0.772399, 1.570796, 1.667924],accel_mss,speed_ms,0,blend_radius_m)
    |   movel([0.095657, -1.333902, -2.605909, -0.772577, 1.570796, 1.666454],accel_mss,speed_ms,0,blend_radius_m)
    |   movel([0.094923, -1.332612, -2.606733, -0.773044, 1.570796, 1.665719],accel_mss,speed_ms,0,blend_radius_m)
    |   movel([0.095096, -1.330833, -2.607866, -0.773690, 1.570796, 1.665892],accel_mss,speed_ms,0,blend_radius_m)
    |   movel([0.096151, -1.328992, -2.609033, -0.774364, 1.570796, 1.666947],accel_mss,speed_ms,0,blend_radius_m)
    |   movel([0.096644, -1.328430, -2.609389, -0.774571, 1.570796, 1.667440],accel_mss,speed_ms,0,blend_radius_m)
    |   movel([0.097190, -1.327882, -2.609734, -0.774772, 1.570796, 1.667986],accel_mss,speed_ms,0,blend_radius_m)
    |   movel([0.097709, -1.327420, -2.610026, -0.774943, 1.570796, 1.668505],accel_mss,speed_ms,0,blend_radius_m)
    |   movel([0.098098, -1.327150, -2.610196, -0.775042, 1.570796, 1.668894],accel_mss,speed_ms,0,blend_radius_m)
    |   movel([0.098496, -1.326850, -2.610385, -0.775153, 1.570796, 1.669292],accel_mss,speed_ms,0,blend_radius_m)
    |   movel([0.098769, -1.326494, -2.610610, -0.775285, 1.570796, 1.669565],accel_mss,speed_ms,0,blend_radius_m)
    |   movel([0.098948, -1.326010, -2.610914, -0.775465, 1.570796, 1.669744],accel_mss,speed_ms,0,blend_radius_m)
    |   movel([0.099064, -1.325301, -2.611359, -0.775728, 1.570796, 1.669860],accel_mss,speed_ms,0,blend_radius_m)
    |   movel([0.099170, -1.324637, -2.611776, -0.775976, 1.570796, 1.669967],accel_mss,speed_ms,0,blend_radius_m)
    |   movel([0.099325, -1.324188, -2.612057, -0.776143, 1.570796, 1.670121],accel_mss,speed_ms,0,blend_radius_m)
    |   movel([0.099542, -1.323896, -2.612241, -0.776253, 1.570796, 1.670338],accel_mss,speed_ms,0,blend_radius_m)
    |   speed_ms = 0.003
    |   movel([0.099542, -1.327369, -2.613818, -0.771202, 1.570796, 1.670338],accel_mss,speed_ms,0,blend_radius_m)
    |   speed_ms = 0.007
    |   movel([0.099826, -1.327197, -2.613926, -0.771266, 1.570796, 1.670622],accel_mss,speed_ms,0,blend_radius_m)
    |   movel([0.100093, -1.327198, -2.613925, -0.771265, 1.570796, 1.670889],accel_mss,speed_ms,0,blend_radius_m)
    |   movel([0.100254, -1.327376, -2.613814, -0.771200, 1.570796, 1.671050],accel_mss,speed_ms,0,blend_radius_m)
    |   movel([0.100313, -1.327764, -2.613569, -0.771056, 1.570796, 1.671109],accel_mss,speed_ms,0,blend_radius_m)
    |   movel([0.100269, -1.328415, -2.613159, -0.770815, 1.570796, 1.671066],accel_mss,speed_ms,0,blend_radius_m)
    |   movel([0.100218, -1.329178, -2.612677, -0.770534, 1.570796, 1.671014],accel_mss,speed_ms,0,blend_radius_m)
    |   movel([0.100312, -1.329552, -2.612441, -0.770396, 1.570796, 1.671108],accel_mss,speed_ms,0,blend_radius_m)
    |   movel([0.100577, -1.329715, -2.612338, -0.770336, 1.570796, 1.671374],accel_mss,speed_ms,0,blend_radius_m)
    |   movel([0.101087, -1.329730, -2.612328, -0.770330, 1.570796, 1.671883],accel_mss,speed_ms,0,blend_radius_m)
    |   movel([0.101527, -1.329747, -2.612318, -0.770324, 1.570796, 1.672323],accel_mss,speed_ms,0,blend_radius_m)
    |   movel([0.102040, -1.329883, -2.612231, -0.770274, 1.570796, 1.672837],accel_mss,speed_ms,0,blend_radius_m)
    |   movel([0.102538, -1.330104, -2.612092, -0.770193, 1.570796, 1.673335],accel_mss,speed_ms,0,blend_radius_m)
    |   movel([0.102947, -1.330380, -2.611917, -0.770092, 1.570796, 1.673743],accel_mss,speed_ms,0,blend_radius_m)
    |   movel([0.103665, -1.331609, -2.611138, -0.769642, 1.570796, 1.674461],accel_mss,speed_ms,0,blend_radius_m)
    |   movel([0.103516, -1.333235, -2.610104, -0.769050, 1.570796, 1.674312],accel_mss,speed_ms,0,blend_radius_m)
    |   movel([0.102517, -1.334977, -2.608991, -0.768420, 1.570796, 1.673313],accel_mss,speed_ms,0,blend_radius_m)
    |   movel([0.100855, -1.336536, -2.607993, -0.767860, 1.570796, 1.671651],accel_mss,speed_ms,0,blend_radius_m)
    |   movel([0.100194, -1.337064, -2.607654, -0.767671, 1.570796, 1.670991],accel_mss,speed_ms,0,blend_radius_m)
    |   movel([0.099818, -1.337509, -2.607368, -0.767512, 1.570796, 1.670614],accel_mss,speed_ms,0,blend_radius_m)
    |   movel([0.099600, -1.338025, -2.607036, -0.767328, 1.570796, 1.670396],accel_mss,speed_ms,0,blend_radius_m)
    |   movel([0.099465, -1.338801, -2.606536, -0.767052, 1.570796, 1.670261],accel_mss,speed_ms,0,blend_radius_m)
    |   movel([0.099351, -1.339550, -2.606053, -0.766786, 1.570796, 1.670148],accel_mss,speed_ms,0,blend_radius_m)
    |   movel([0.099189, -1.339965, -2.605785, -0.766640, 1.570796, 1.669985],accel_mss,speed_ms,0,blend_radius_m)
    |   movel([0.098926, -1.340229, -2.605614, -0.766546, 1.570796, 1.669723],accel_mss,speed_ms,0,blend_radius_m)
    |   movel([0.098514, -1.340419, -2.605491, -0.766479, 1.570796, 1.669311],accel_mss,speed_ms,0,blend_radius_m)
    |   movel([0.098117, -1.340473, -2.605456, -0.766460, 1.570796, 1.668914],accel_mss,speed_ms,0,blend_radius_m)
    |   movel([0.097898, -1.340355, -2.605533, -0.766502, 1.570796, 1.668695],accel_mss,speed_ms,0,blend_radius_m)
    |   movel([0.097822, -1.340008, -2.605757, -0.766624, 1.570796, 1.668619],accel_mss,speed_ms,0,blend_radius_m)
    |   movel([0.097878, -1.339266, -2.606236, -0.766887, 1.570796, 1.668674],accel_mss,speed_ms,0,blend_radius_m)
    |   movel([0.097922, -1.338534, -2.606708, -0.767147, 1.570796, 1.668718],accel_mss,speed_ms,0,blend_radius_m)
    |   movel([0.097831, -1.338133, -2.606967, -0.767290, 1.570796, 1.668627],accel_mss,speed_ms,0,blend_radius_m)
    |   movel([0.097583, -1.337925, -2.607100, -0.767364, 1.570796, 1.668379],accel_mss,speed_ms,0,blend_radius_m)
    |   movel([0.097128, -1.337845, -2.607152, -0.767392, 1.570796, 1.667924],accel_mss,speed_ms,0,blend_radius_m)
    |   movel([0.095657, -1.337350, -2.607470, -0.767569, 1.570796, 1.666454],accel_mss,speed_ms,0,blend_radius_m)
    |   movel([0.094923, -1.336063, -2.608296, -0.768030, 1.570796, 1.665719],accel_mss,speed_ms,0,blend_radius_m)
    |   movel([0.095096, -1.334289, -2.609431, -0.768669, 1.570796, 1.665892],accel_mss,speed_ms,0,blend_radius_m)
    |   movel([0.096151, -1.332452, -2.610602, -0.769335, 1.570796, 1.666947],accel_mss,speed_ms,0,blend_radius_m)
    |   movel([0.096644, -1.331892, -2.610958, -0.769539, 1.570796, 1.667440],accel_mss,speed_ms,0,blend_radius_m)
    |   movel([0.097190, -1.331346, -2.611305, -0.769738, 1.570796, 1.667986],accel_mss,speed_ms,0,blend_radius_m)
    |   movel([0.097709, -1.330885, -2.611597, -0.769907, 1.570796, 1.668505],accel_mss,speed_ms,0,blend_radius_m)
    |   movel([0.098098, -1.330615, -2.611768, -0.770006, 1.570796, 1.668894],accel_mss,speed_ms,0,blend_radius_m)
    |   movel([0.098496, -1.330316, -2.611958, -0.770115, 1.570796, 1.669292],accel_mss,speed_ms,0,blend_radius_m)
    |   movel([0.098769, -1.329960, -2.612183, -0.770246, 1.570796, 1.669565],accel_mss,speed_ms,0,blend_radius_m)
    |   movel([0.098948, -1.329477, -2.612488, -0.770423, 1.570796, 1.669744],accel_mss,speed_ms,0,blend_radius_m)
    |   movel([0.099064, -1.328771, -2.612934, -0.770684, 1.570796, 1.669860],accel_mss,speed_ms,0,blend_radius_m)
    |   movel([0.099170, -1.328108, -2.613352, -0.770928, 1.570796, 1.669967],accel_mss,speed_ms,0,blend_radius_m)
    |   movel([0.099325, -1.327661, -2.613634, -0.771094, 1.570796, 1.670121],accel_mss,speed_ms,0,blend_radius_m)
    |   movel([0.099542, -1.327369, -2.613818, -0.771202, 1.570796, 1.670338],accel_mss,speed_ms,0,blend_radius_m)
    |   speed_ms = 0.003
    |   # Splitting Linear movement in 6 (instruction 283: MoveL 261)
    |   movel([0.099542, -1.325050, -2.612767, -0.774571, 1.570796, 1.670338],accel_mss,speed_ms,0,blend_radius_m)
    |   movel([0.099542, -1.322744, -2.611713, -0.777932, 1.570796, 1.670338],accel_mss,speed_ms,0,blend_radius_m)
    |   movel([0.099542, -1.320449, -2.610655, -0.781285, 1.570796, 1.670338],accel_mss,speed_ms,0,blend_radius_m)
    |   movel([0.099542, -1.318166, -2.609593, -0.784630, 1.570796, 1.670338],accel_mss,speed_ms,0,blend_radius_m)
    |   movel([0.099542, -1.315894, -2.608527, -0.787967, 1.570796, 1.670338],accel_mss,speed_ms,0,blend_radius_m)
    |   movel([0.099542, -1.313635, -2.607458, -0.791296, 1.570796, 1.670338],accel_mss,speed_ms,0,blend_radius_m)
    |   speed_ms = 1.000
    |   # Splitting Linear movement in 12 (instruction 285: MoveL 262)
    |   movel([0.099542, -1.311387, -2.606385, -0.794617, 1.570796, 1.670338],accel_mss,speed_ms,0,blend_radius_m)
    |   movel([0.099542, -1.309150, -2.605309, -0.797930, 1.570796, 1.670338],accel_mss,speed_ms,0,blend_radius_m)
    |   movel([0.099542, -1.306925, -2.604228, -0.801235, 1.570796, 1.670338],accel_mss,speed_ms,0,blend_radius_m)
    |   movel([0.099542, -1.304712, -2.603145, -0.804532, 1.570796, 1.670338],accel_mss,speed_ms,0,blend_radius_m)
    |   movel([0.099542, -1.302511, -2.602057, -0.807821, 1.570796, 1.670338],accel_mss,speed_ms,0,blend_radius_m)
    |   movel([0.099542, -1.300321, -2.600966, -0.811102, 1.570796, 1.670338],accel_mss,speed_ms,0,blend_radius_m)
    |   movel([0.099542, -1.298142, -2.599872, -0.814375, 1.570796, 1.670338],accel_mss,speed_ms,0,blend_radius_m)
    |   movel([0.099542, -1.295975, -2.598774, -0.817641, 1.570796, 1.670338],accel_mss,speed_ms,0,blend_radius_m)
    |   movel([0.099542, -1.293819, -2.597672, -0.820898, 1.570796, 1.670338],accel_mss,speed_ms,0,blend_radius_m)
    |   movel([0.099542, -1.291675, -2.596567, -0.824147, 1.570796, 1.670338],accel_mss,speed_ms,0,blend_radius_m)
    |   movel([0.099542, -1.289542, -2.595458, -0.827389, 1.570796, 1.670338],accel_mss,speed_ms,0,blend_radius_m)
    |   movel([0.099542, -1.287421, -2.594346, -0.830622, 1.570796, 1.670338],accel_mss,speed_ms,0,blend_radius_m)
    |   # Splitting Linear movement in 6 (instruction 286: MoveL 263)
    |   movel([0.101356, -1.287568, -2.594259, -0.830563, 1.570796, 1.672152],accel_mss,speed_ms,0,blend_radius_m)
    |   movel([0.103168, -1.287718, -2.594169, -0.830502, 1.570796, 1.673964],accel_mss,speed_ms,0,blend_radius_m)
    |   movel([0.104978, -1.287872, -2.594078, -0.830439, 1.570796, 1.675774],accel_mss,speed_ms,0,blend_radius_m)
    |   movel([0.106785, -1.288030, -2.593984, -0.830375, 1.570796, 1.677582],accel_mss,speed_ms,0,blend_radius_m)
    |   movel([0.108591, -1.288191, -2.593888, -0.830310, 1.570796, 1.679387],accel_mss,speed_ms,0,blend_radius_m)
    |   movel([0.110394, -1.288356, -2.593790, -0.830243, 1.570796, 1.681190],accel_mss,speed_ms,0,blend_radius_m)
    |   # Splitting Linear movement in 14 (instruction 287: MoveL 264)
    |   movel([0.110394, -1.290173, -2.594742, -0.827474, 1.570796, 1.681190],accel_mss,speed_ms,0,blend_radius_m)
    |   movel([0.110394, -1.291998, -2.595692, -0.824698, 1.570796, 1.681190],accel_mss,speed_ms,0,blend_radius_m)
    |   movel([0.110394, -1.293832, -2.596640, -0.821917, 1.570796, 1.681190],accel_mss,speed_ms,0,blend_radius_m)
    |   movel([0.110394, -1.295674, -2.597585, -0.819131, 1.570796, 1.681190],accel_mss,speed_ms,0,blend_radius_m)
    |   movel([0.110394, -1.297524, -2.598527, -0.816338, 1.570796, 1.681190],accel_mss,speed_ms,0,blend_radius_m)
    |   movel([0.110394, -1.299382, -2.599467, -0.813540, 1.570796, 1.681190],accel_mss,speed_ms,0,blend_radius_m)
    |   movel([0.110394, -1.301249, -2.600404, -0.810736, 1.570796, 1.681190],accel_mss,speed_ms,0,blend_radius_m)
    |   movel([0.110394, -1.303125, -2.601338, -0.807926, 1.570796, 1.681190],accel_mss,speed_ms,0,blend_radius_m)
    |   movel([0.110394, -1.305009, -2.602270, -0.805110, 1.570796, 1.681190],accel_mss,speed_ms,0,blend_radius_m)
    |   movel([0.110394, -1.306901, -2.603199, -0.802288, 1.570796, 1.681190],accel_mss,speed_ms,0,blend_radius_m)
    |   movel([0.110394, -1.308802, -2.604126, -0.799461, 1.570796, 1.681190],accel_mss,speed_ms,0,blend_radius_m)
    |   movel([0.110394, -1.310712, -2.605050, -0.796628, 1.570796, 1.681190],accel_mss,speed_ms,0,blend_radius_m)
    |   movel([0.110394, -1.312630, -2.605971, -0.793788, 1.570796, 1.681190],accel_mss,speed_ms,0,blend_radius_m)
    |   movel([0.110394, -1.314556, -2.606890, -0.790943, 1.570796, 1.681190],accel_mss,speed_ms,0,blend_radius_m)
    |   speed_ms = 0.003
    |   # Splitting Linear movement in 6 (instruction 289: MoveL 265)
    |   movel([0.110394, -1.316249, -2.607691, -0.788449, 1.570796, 1.681190],accel_mss,speed_ms,0,blend_radius_m)
    |   movel([0.110394, -1.317948, -2.608491, -0.785951, 1.570796, 1.681190],accel_mss,speed_ms,0,blend_radius_m)
    |   movel([0.110394, -1.319654, -2.609288, -0.783447, 1.570796, 1.681190],accel_mss,speed_ms,0,blend_radius_m)
    |   movel([0.110394, -1.321366, -2.610083, -0.780940, 1.570796, 1.681190],accel_mss,speed_ms,0,blend_radius_m)
    |   movel([0.110394, -1.323085, -2.610876, -0.778428, 1.570796, 1.681190],accel_mss,speed_ms,0,blend_radius_m)
    |   movel([0.110394, -1.324811, -2.611667, -0.775911, 1.570796, 1.681190],accel_mss,speed_ms,0,blend_radius_m)
    |   speed_ms = 0.007
    |   movel([0.112438, -1.322918, -2.612852, -0.776619, 1.570796, 1.683234],accel_mss,speed_ms,0,blend_radius_m)
    |   movel([0.112923, -1.322555, -2.613079, -0.776755, 1.570796, 1.683719],accel_mss,speed_ms,0,blend_radius_m)
    |   movel([0.113236, -1.322171, -2.613318, -0.776900, 1.570796, 1.684032],accel_mss,speed_ms,0,blend_radius_m)
    |   movel([0.113432, -1.321671, -2.613630, -0.777088, 1.570796, 1.684229],accel_mss,speed_ms,0,blend_radius_m)
    |   movel([0.113570, -1.320904, -2.614107, -0.777378, 1.570796, 1.684366],accel_mss,speed_ms,0,blend_radius_m)
    |   movel([0.113699, -1.320121, -2.614594, -0.777674, 1.570796, 1.684496],accel_mss,speed_ms,0,blend_radius_m)
    |   movel([0.113872, -1.319689, -2.614862, -0.777838, 1.570796, 1.684668],accel_mss,speed_ms,0,blend_radius_m)
    |   movel([0.114143, -1.319417, -2.615031, -0.777941, 1.570796, 1.684939],accel_mss,speed_ms,0,blend_radius_m)
    |   movel([0.114565, -1.319221, -2.615152, -0.778016, 1.570796, 1.685361],accel_mss,speed_ms,0,blend_radius_m)
    |   movel([0.114968, -1.319166, -2.615186, -0.778037, 1.570796, 1.685764],accel_mss,speed_ms,0,blend_radius_m)
    |   movel([0.115185, -1.319289, -2.615110, -0.777990, 1.570796, 1.685982],accel_mss,speed_ms,0,blend_radius_m)
    |   movel([0.115258, -1.319642, -2.614891, -0.777856, 1.570796, 1.686055],accel_mss,speed_ms,0,blend_radius_m)
    |   movel([0.115190, -1.320387, -2.614429, -0.777573, 1.570796, 1.685986],accel_mss,speed_ms,0,blend_radius_m)
    |   movel([0.115135, -1.321081, -2.613997, -0.777311, 1.570796, 1.685931],accel_mss,speed_ms,0,blend_radius_m)
    |   movel([0.115205, -1.321492, -2.613741, -0.777155, 1.570796, 1.686002],accel_mss,speed_ms,0,blend_radius_m)
    |   movel([0.115410, -1.321706, -2.613608, -0.777075, 1.570796, 1.686206],accel_mss,speed_ms,0,blend_radius_m)
    |   movel([0.115765, -1.321778, -2.613563, -0.777048, 1.570796, 1.686561],accel_mss,speed_ms,0,blend_radius_m)
    |   movel([0.116118, -1.321824, -2.613534, -0.777030, 1.570796, 1.686914],accel_mss,speed_ms,0,blend_radius_m)
    |   movel([0.116562, -1.321996, -2.613427, -0.776966, 1.570796, 1.687359],accel_mss,speed_ms,0,blend_radius_m)
    |   movel([0.117015, -1.322244, -2.613273, -0.776872, 1.570796, 1.687811],accel_mss,speed_ms,0,blend_radius_m)
    |   movel([0.117406, -1.322541, -2.613087, -0.776761, 1.570796, 1.688203],accel_mss,speed_ms,0,blend_radius_m)
    |   movel([0.118081, -1.323873, -2.612255, -0.776261, 1.570796, 1.688878],accel_mss,speed_ms,0,blend_radius_m)
    |   movel([0.117817, -1.325698, -2.611110, -0.775581, 1.570796, 1.688613],accel_mss,speed_ms,0,blend_radius_m)
    |   movel([0.116693, -1.327565, -2.609935, -0.774889, 1.570796, 1.687489],accel_mss,speed_ms,0,blend_radius_m)
    |   movel([0.114974, -1.329029, -2.609010, -0.774350, 1.570796, 1.685770],accel_mss,speed_ms,0,blend_radius_m)
    |   movel([0.114462, -1.329402, -2.608774, -0.774214, 1.570796, 1.685258],accel_mss,speed_ms,0,blend_radius_m)
    |   movel([0.114140, -1.329784, -2.608532, -0.774074, 1.570796, 1.684937],accel_mss,speed_ms,0,blend_radius_m)
    |   movel([0.113941, -1.330276, -2.608219, -0.773894, 1.570796, 1.684737],accel_mss,speed_ms,0,blend_radius_m)
    |   movel([0.113803, -1.331044, -2.607732, -0.773613, 1.570796, 1.684599],accel_mss,speed_ms,0,blend_radius_m)
    |   movel([0.113687, -1.331723, -2.607300, -0.773366, 1.570796, 1.684483],accel_mss,speed_ms,0,blend_radius_m)
    |   movel([0.113526, -1.332176, -2.607011, -0.773202, 1.570796, 1.684322],accel_mss,speed_ms,0,blend_radius_m)
    |   movel([0.113307, -1.332465, -2.606827, -0.773097, 1.570796, 1.684103],accel_mss,speed_ms,0,blend_radius_m)
    |   movel([0.113022, -1.332635, -2.606719, -0.773035, 1.570796, 1.683819],accel_mss,speed_ms,0,blend_radius_m)
    |   movel([0.112762, -1.332630, -2.606722, -0.773037, 1.570796, 1.683559],accel_mss,speed_ms,0,blend_radius_m)
    |   movel([0.112603, -1.332459, -2.606831, -0.773099, 1.570796, 1.683399],accel_mss,speed_ms,0,blend_radius_m)
    |   movel([0.112548, -1.332088, -2.607068, -0.773234, 1.570796, 1.683345],accel_mss,speed_ms,0,blend_radius_m)
    |   movel([0.112597, -1.331472, -2.607460, -0.773458, 1.570796, 1.683393],accel_mss,speed_ms,0,blend_radius_m)
    |   movel([0.112644, -1.330722, -2.607936, -0.773731, 1.570796, 1.683440],accel_mss,speed_ms,0,blend_radius_m)
    |   movel([0.112518, -1.330329, -2.608186, -0.773874, 1.570796, 1.683314],accel_mss,speed_ms,0,blend_radius_m)
    |   movel([0.112178, -1.330102, -2.608330, -0.773957, 1.570796, 1.682974],accel_mss,speed_ms,0,blend_radius_m)
    |   movel([0.111464, -1.329957, -2.608422, -0.774010, 1.570796, 1.682260],accel_mss,speed_ms,0,blend_radius_m)
    |   movel([0.109809, -1.329045, -2.609000, -0.774345, 1.570796, 1.680605],accel_mss,speed_ms,0,blend_radius_m)
    |   movel([0.109408, -1.327111, -2.610221, -0.775057, 1.570796, 1.680204],accel_mss,speed_ms,0,blend_radius_m)
    |   movel([0.110394, -1.324811, -2.611667, -0.775911, 1.570796, 1.681190],accel_mss,speed_ms,0,blend_radius_m)
    |   speed_ms = 0.003
    |   movel([0.110394, -1.328281, -2.613243, -0.770864, 1.570796, 1.681190],accel_mss,speed_ms,0,blend_radius_m)
    |   speed_ms = 0.007
    |   movel([0.112438, -1.326393, -2.614431, -0.771565, 1.570796, 1.683234],accel_mss,speed_ms,0,blend_radius_m)
    |   movel([0.112923, -1.326032, -2.614658, -0.771699, 1.570796, 1.683719],accel_mss,speed_ms,0,blend_radius_m)
    |   movel([0.113236, -1.325649, -2.614898, -0.771842, 1.570796, 1.684032],accel_mss,speed_ms,0,blend_radius_m)
    |   movel([0.113432, -1.325150, -2.615211, -0.772028, 1.570796, 1.684229],accel_mss,speed_ms,0,blend_radius_m)
    |   movel([0.113570, -1.324385, -2.615689, -0.772315, 1.570796, 1.684366],accel_mss,speed_ms,0,blend_radius_m)
    |   movel([0.113699, -1.323603, -2.616178, -0.772608, 1.570796, 1.684496],accel_mss,speed_ms,0,blend_radius_m)
    |   movel([0.113872, -1.323172, -2.616447, -0.772770, 1.570796, 1.684668],accel_mss,speed_ms,0,blend_radius_m)
    |   movel([0.114143, -1.322901, -2.616616, -0.772872, 1.570796, 1.684939],accel_mss,speed_ms,0,blend_radius_m)
    |   movel([0.114565, -1.322706, -2.616737, -0.772946, 1.570796, 1.685361],accel_mss,speed_ms,0,blend_radius_m)
    |   movel([0.114968, -1.322651, -2.616771, -0.772966, 1.570796, 1.685764],accel_mss,speed_ms,0,blend_radius_m)
    |   movel([0.115185, -1.322774, -2.616695, -0.772920, 1.570796, 1.685982],accel_mss,speed_ms,0,blend_radius_m)
    |   movel([0.115258, -1.323125, -2.616476, -0.772788, 1.570796, 1.686055],accel_mss,speed_ms,0,blend_radius_m)
    |   movel([0.115190, -1.323868, -2.616012, -0.772508, 1.570796, 1.685986],accel_mss,speed_ms,0,blend_radius_m)
    |   movel([0.115135, -1.324561, -2.615579, -0.772249, 1.570796, 1.685931],accel_mss,speed_ms,0,blend_radius_m)
    |   movel([0.115205, -1.324972, -2.615322, -0.772095, 1.570796, 1.686002],accel_mss,speed_ms,0,blend_radius_m)
    |   movel([0.115410, -1.325184, -2.615189, -0.772015, 1.570796, 1.686206],accel_mss,speed_ms,0,blend_radius_m)
    |   movel([0.115765, -1.325257, -2.615144, -0.771988, 1.570796, 1.686561],accel_mss,speed_ms,0,blend_radius_m)
    |   movel([0.116118, -1.325303, -2.615115, -0.771971, 1.570796, 1.686914],accel_mss,speed_ms,0,blend_radius_m)
    |   movel([0.116562, -1.325474, -2.615008, -0.771907, 1.570796, 1.687359],accel_mss,speed_ms,0,blend_radius_m)
    |   movel([0.117015, -1.325721, -2.614853, -0.771815, 1.570796, 1.687811],accel_mss,speed_ms,0,blend_radius_m)
    |   movel([0.117406, -1.326018, -2.614667, -0.771704, 1.570796, 1.688203],accel_mss,speed_ms,0,blend_radius_m)
    |   movel([0.118081, -1.327347, -2.613832, -0.771210, 1.570796, 1.688878],accel_mss,speed_ms,0,blend_radius_m)
    |   movel([0.117817, -1.329167, -2.612684, -0.770538, 1.570796, 1.688613],accel_mss,speed_ms,0,blend_radius_m)
    |   movel([0.116693, -1.331029, -2.611506, -0.769854, 1.570796, 1.687489],accel_mss,speed_ms,0,blend_radius_m)
    |   movel([0.114974, -1.332489, -2.610578, -0.769321, 1.570796, 1.685770],accel_mss,speed_ms,0,blend_radius_m)
    |   movel([0.114462, -1.332861, -2.610342, -0.769186, 1.570796, 1.685258],accel_mss,speed_ms,0,blend_radius_m)
    |   movel([0.114140, -1.333242, -2.610099, -0.769048, 1.570796, 1.684937],accel_mss,speed_ms,0,blend_radius_m)
    |   movel([0.113941, -1.333734, -2.609786, -0.768870, 1.570796, 1.684737],accel_mss,speed_ms,0,blend_radius_m)
    |   movel([0.113803, -1.334499, -2.609297, -0.768593, 1.570796, 1.684599],accel_mss,speed_ms,0,blend_radius_m)
    |   movel([0.113687, -1.335177, -2.608864, -0.768349, 1.570796, 1.684483],accel_mss,speed_ms,0,blend_radius_m)
    |   movel([0.113526, -1.335628, -2.608575, -0.768186, 1.570796, 1.684322],accel_mss,speed_ms,0,blend_radius_m)
    |   movel([0.113307, -1.335917, -2.608390, -0.768082, 1.570796, 1.684103],accel_mss,speed_ms,0,blend_radius_m)
    |   movel([0.113022, -1.336086, -2.608281, -0.768021, 1.570796, 1.683819],accel_mss,speed_ms,0,blend_radius_m)
    |   movel([0.112762, -1.336082, -2.608284, -0.768023, 1.570796, 1.683559],accel_mss,speed_ms,0,blend_radius_m)
    |   movel([0.112603, -1.335911, -2.608394, -0.768084, 1.570796, 1.683399],accel_mss,speed_ms,0,blend_radius_m)
    |   movel([0.112548, -1.335540, -2.608631, -0.768218, 1.570796, 1.683345],accel_mss,speed_ms,0,blend_radius_m)
    |   movel([0.112597, -1.334926, -2.609024, -0.768439, 1.570796, 1.683393],accel_mss,speed_ms,0,blend_radius_m)
    |   movel([0.112644, -1.334179, -2.609502, -0.768709, 1.570796, 1.683440],accel_mss,speed_ms,0,blend_radius_m)
    |   movel([0.112518, -1.333786, -2.609752, -0.768851, 1.570796, 1.683314],accel_mss,speed_ms,0,blend_radius_m)
    |   movel([0.112178, -1.333560, -2.609897, -0.768933, 1.570796, 1.682974],accel_mss,speed_ms,0,blend_radius_m)
    |   movel([0.111464, -1.333415, -2.609989, -0.768985, 1.570796, 1.682260],accel_mss,speed_ms,0,blend_radius_m)
    |   movel([0.109809, -1.332505, -2.610568, -0.769316, 1.570796, 1.680605],accel_mss,speed_ms,0,blend_radius_m)
    |   movel([0.109408, -1.330576, -2.611793, -0.770020, 1.570796, 1.680204],accel_mss,speed_ms,0,blend_radius_m)
    |   movel([0.110394, -1.328281, -2.613243, -0.770864, 1.570796, 1.681190],accel_mss,speed_ms,0,blend_radius_m)
    |   speed_ms = 0.003
    |   # Splitting Linear movement in 6 (instruction 383: MoveL 355)
    |   movel([0.110394, -1.325965, -2.612194, -0.774231, 1.570796, 1.681190],accel_mss,speed_ms,0,blend_radius_m)
    |   movel([0.110394, -1.323659, -2.611140, -0.777589, 1.570796, 1.681190],accel_mss,speed_ms,0,blend_radius_m)
    |   movel([0.110394, -1.321366, -2.610083, -0.780940, 1.570796, 1.681190],accel_mss,speed_ms,0,blend_radius_m)
    |   movel([0.110394, -1.319084, -2.609022, -0.784282, 1.570796, 1.681190],accel_mss,speed_ms,0,blend_radius_m)
    |   movel([0.110394, -1.316814, -2.607958, -0.787617, 1.570796, 1.681190],accel_mss,speed_ms,0,blend_radius_m)
    |   movel([0.110394, -1.314556, -2.606890, -0.790943, 1.570796, 1.681190],accel_mss,speed_ms,0,blend_radius_m)
    |   speed_ms = 1.000
    |   # Splitting Linear movement in 14 (instruction 385: MoveL 356)
    |   movel([0.110394, -1.312630, -2.605971, -0.793788, 1.570796, 1.681190],accel_mss,speed_ms,0,blend_radius_m)
    |   movel([0.110394, -1.310712, -2.605050, -0.796628, 1.570796, 1.681190],accel_mss,speed_ms,0,blend_radius_m)
    |   movel([0.110394, -1.308802, -2.604126, -0.799461, 1.570796, 1.681190],accel_mss,speed_ms,0,blend_radius_m)
    |   movel([0.110394, -1.306901, -2.603199, -0.802288, 1.570796, 1.681190],accel_mss,speed_ms,0,blend_radius_m)
    |   movel([0.110394, -1.305009, -2.602270, -0.805110, 1.570796, 1.681190],accel_mss,speed_ms,0,blend_radius_m)
    |   movel([0.110394, -1.303125, -2.601338, -0.807926, 1.570796, 1.681190],accel_mss,speed_ms,0,blend_radius_m)
    |   movel([0.110394, -1.301249, -2.600404, -0.810736, 1.570796, 1.681190],accel_mss,speed_ms,0,blend_radius_m)
    |   movel([0.110394, -1.299382, -2.599467, -0.813540, 1.570796, 1.681190],accel_mss,speed_ms,0,blend_radius_m)
    |   movel([0.110394, -1.297524, -2.598527, -0.816338, 1.570796, 1.681190],accel_mss,speed_ms,0,blend_radius_m)
    |   movel([0.110394, -1.295674, -2.597585, -0.819131, 1.570796, 1.681190],accel_mss,speed_ms,0,blend_radius_m)
    |   movel([0.110394, -1.293832, -2.596640, -0.821917, 1.570796, 1.681190],accel_mss,speed_ms,0,blend_radius_m)
    |   movel([0.110394, -1.291998, -2.595692, -0.824698, 1.570796, 1.681190],accel_mss,speed_ms,0,blend_radius_m)
    |   movel([0.110394, -1.290173, -2.594742, -0.827474, 1.570796, 1.681190],accel_mss,speed_ms,0,blend_radius_m)
    |   movel([0.110394, -1.288356, -2.593790, -0.830243, 1.570796, 1.681190],accel_mss,speed_ms,0,blend_radius_m)
    |   # Splitting Linear movement in 6 (instruction 386: MoveL 357)
    |   movel([0.112644, -1.288050, -2.593972, -0.830367, 1.570796, 1.683440],accel_mss,speed_ms,0,blend_radius_m)
    |   movel([0.114894, -1.287747, -2.594152, -0.830490, 1.570796, 1.685690],accel_mss,speed_ms,0,blend_radius_m)
    |   movel([0.117142, -1.287450, -2.594329, -0.830611, 1.570796, 1.687939],accel_mss,speed_ms,0,blend_radius_m)
    |   movel([0.119390, -1.287156, -2.594503, -0.830730, 1.570796, 1.690187],accel_mss,speed_ms,0,blend_radius_m)
    |   movel([0.121638, -1.286868, -2.594674, -0.830847, 1.570796, 1.692434],accel_mss,speed_ms,0,blend_radius_m)
    |   movel([0.123884, -1.286584, -2.594843, -0.830963, 1.570796, 1.694680],accel_mss,speed_ms,0,blend_radius_m)
    |   # Splitting Linear movement in 12 (instruction 387: MoveL 358)
    |   movel([0.123884, -1.288706, -2.595956, -0.827727, 1.570796, 1.694680],accel_mss,speed_ms,0,blend_radius_m)
    |   movel([0.123884, -1.290840, -2.597065, -0.824484, 1.570796, 1.694680],accel_mss,speed_ms,0,blend_radius_m)
    |   movel([0.123884, -1.292985, -2.598171, -0.821233, 1.570796, 1.694680],accel_mss,speed_ms,0,blend_radius_m)
    |   movel([0.123884, -1.295142, -2.599274, -0.817973, 1.570796, 1.694680],accel_mss,speed_ms,0,blend_radius_m)
    |   movel([0.123884, -1.297310, -2.600373, -0.814706, 1.570796, 1.694680],accel_mss,speed_ms,0,blend_radius_m)
    |   movel([0.123884, -1.299489, -2.601468, -0.811431, 1.570796, 1.694680],accel_mss,speed_ms,0,blend_radius_m)
    |   movel([0.123884, -1.301681, -2.602560, -0.808148, 1.570796, 1.694680],accel_mss,speed_ms,0,blend_radius_m)
    |   movel([0.123884, -1.303883, -2.603649, -0.804857, 1.570796, 1.694680],accel_mss,speed_ms,0,blend_radius_m)
    |   movel([0.123884, -1.306098, -2.604734, -0.801558, 1.570796, 1.694680],accel_mss,speed_ms,0,blend_radius_m)
    |   movel([0.123884, -1.308324, -2.605815, -0.798251, 1.570796, 1.694680],accel_mss,speed_ms,0,blend_radius_m)
    |   movel([0.123884, -1.310561, -2.606892, -0.794936, 1.570796, 1.694680],accel_mss,speed_ms,0,blend_radius_m)
    |   movel([0.123884, -1.312811, -2.607966, -0.791612, 1.570796, 1.694680],accel_mss,speed_ms,0,blend_radius_m)
    |   speed_ms = 0.003
    |   # Splitting Linear movement in 6 (instruction 389: MoveL 359)
    |   movel([0.123884, -1.314505, -2.608769, -0.789115, 1.570796, 1.694680],accel_mss,speed_ms,0,blend_radius_m)
    |   movel([0.123884, -1.316206, -2.609570, -0.786613, 1.570796, 1.694680],accel_mss,speed_ms,0,blend_radius_m)
    |   movel([0.123884, -1.317914, -2.610369, -0.784106, 1.570796, 1.694680],accel_mss,speed_ms,0,blend_radius_m)
    |   movel([0.123884, -1.319629, -2.611165, -0.781595, 1.570796, 1.694680],accel_mss,speed_ms,0,blend_radius_m)
    |   movel([0.123884, -1.321350, -2.611960, -0.779079, 1.570796, 1.694680],accel_mss,speed_ms,0,blend_radius_m)
    |   movel([0.123884, -1.323077, -2.612753, -0.776559, 1.570796, 1.694680],accel_mss,speed_ms,0,blend_radius_m)
    |   speed_ms = 0.007
    |   movel([0.124792, -1.320870, -2.614128, -0.777390, 1.570796, 1.695588],accel_mss,speed_ms,0,blend_radius_m)
    |   movel([0.126733, -1.318901, -2.615351, -0.778138, 1.570796, 1.697529],accel_mss,speed_ms,0,blend_radius_m)
    |   movel([0.127638, -1.318208, -2.615779, -0.778402, 1.570796, 1.698435],accel_mss,speed_ms,0,blend_radius_m)
    |   movel([0.128111, -1.317709, -2.616087, -0.778592, 1.570796, 1.698907],accel_mss,speed_ms,0,blend_radius_m)
    |   movel([0.128379, -1.317175, -2.616417, -0.778797, 1.570796, 1.699175],accel_mss,speed_ms,0,blend_radius_m)
    |   movel([0.128550, -1.316387, -2.616903, -0.779099, 1.570796, 1.699347],accel_mss,speed_ms,0,blend_radius_m)
    |   movel([0.128674, -1.315746, -2.617298, -0.779345, 1.570796, 1.699471],accel_mss,speed_ms,0,blend_radius_m)
    |   movel([0.128842, -1.315305, -2.617569, -0.779515, 1.570796, 1.699638],accel_mss,speed_ms,0,blend_radius_m)
    |   movel([0.129067, -1.315019, -2.617744, -0.779625, 1.570796, 1.699864],accel_mss,speed_ms,0,blend_radius_m)
    |   movel([0.129356, -1.314852, -2.617847, -0.779690, 1.570796, 1.700152],accel_mss,speed_ms,0,blend_radius_m)
    |   movel([0.129619, -1.314859, -2.617843, -0.779687, 1.570796, 1.700416],accel_mss,speed_ms,0,blend_radius_m)
    |   movel([0.129777, -1.315038, -2.617733, -0.779618, 1.570796, 1.700573],accel_mss,speed_ms,0,blend_radius_m)
    |   movel([0.129825, -1.315422, -2.617497, -0.779470, 1.570796, 1.700621],accel_mss,speed_ms,0,blend_radius_m)
    |   movel([0.129763, -1.316057, -2.617106, -0.779226, 1.570796, 1.700559],accel_mss,speed_ms,0,blend_radius_m)
    |   movel([0.129702, -1.316830, -2.616630, -0.778929, 1.570796, 1.700498],accel_mss,speed_ms,0,blend_radius_m)
    |   movel([0.129820, -1.317238, -2.616378, -0.778772, 1.570796, 1.700617],accel_mss,speed_ms,0,blend_radius_m)
    |   movel([0.130166, -1.317473, -2.616233, -0.778683, 1.570796, 1.700962],accel_mss,speed_ms,0,blend_radius_m)
    |   movel([0.130909, -1.317635, -2.616133, -0.778621, 1.570796, 1.701705],accel_mss,speed_ms,0,blend_radius_m)
    |   movel([0.131488, -1.317784, -2.616041, -0.778564, 1.570796, 1.702285],accel_mss,speed_ms,0,blend_radius_m)
    |   movel([0.131996, -1.318051, -2.615876, -0.778461, 1.570796, 1.702792],accel_mss,speed_ms,0,blend_radius_m)
    |   movel([0.132396, -1.318414, -2.615652, -0.778323, 1.570796, 1.703192],accel_mss,speed_ms,0,blend_radius_m)
    |   movel([0.132649, -1.318841, -2.615387, -0.778160, 1.570796, 1.703446],accel_mss,speed_ms,0,blend_radius_m)
    |   movel([0.132924, -1.319711, -2.614849, -0.777830, 1.570796, 1.703720],accel_mss,speed_ms,0,blend_radius_m)
    |   movel([0.132947, -1.320343, -2.614456, -0.777590, 1.570796, 1.703744],accel_mss,speed_ms,0,blend_radius_m)
    |   movel([0.132731, -1.321049, -2.614017, -0.777323, 1.570796, 1.703527],accel_mss,speed_ms,0,blend_radius_m)
    |   movel([0.132168, -1.322167, -2.613321, -0.776901, 1.570796, 1.702965],accel_mss,speed_ms,0,blend_radius_m)
    |   movel([0.131743, -1.322833, -2.612905, -0.776651, 1.570796, 1.702540],accel_mss,speed_ms,0,blend_radius_m)
    |   movel([0.131210, -1.323471, -2.612506, -0.776412, 1.570796, 1.702006],accel_mss,speed_ms,0,blend_radius_m)
    |   movel([0.130584, -1.324060, -2.612138, -0.776191, 1.570796, 1.701380],accel_mss,speed_ms,0,blend_radius_m)
    |   movel([0.129887, -1.324583, -2.611810, -0.775996, 1.570796, 1.700683],accel_mss,speed_ms,0,blend_radius_m)
    |   movel([0.129036, -1.325197, -2.611425, -0.775767, 1.570796, 1.699832],accel_mss,speed_ms,0,blend_radius_m)
    |   movel([0.128593, -1.325653, -2.611138, -0.775597, 1.570796, 1.699389],accel_mss,speed_ms,0,blend_radius_m)
    |   movel([0.128342, -1.326162, -2.610819, -0.775409, 1.570796, 1.699139],accel_mss,speed_ms,0,blend_radius_m)
    |   movel([0.128176, -1.326953, -2.610321, -0.775115, 1.570796, 1.698973],accel_mss,speed_ms,0,blend_radius_m)
    |   movel([0.128053, -1.327595, -2.609916, -0.774878, 1.570796, 1.698849],accel_mss,speed_ms,0,blend_radius_m)
    |   movel([0.127887, -1.328032, -2.609640, -0.774717, 1.570796, 1.698683],accel_mss,speed_ms,0,blend_radius_m)
    |   movel([0.127665, -1.328316, -2.609461, -0.774613, 1.570796, 1.698461],accel_mss,speed_ms,0,blend_radius_m)
    |   movel([0.127381, -1.328478, -2.609358, -0.774553, 1.570796, 1.698177],accel_mss,speed_ms,0,blend_radius_m)
    |   movel([0.127121, -1.328470, -2.609363, -0.774556, 1.570796, 1.697918],accel_mss,speed_ms,0,blend_radius_m)
    |   movel([0.126965, -1.328295, -2.609474, -0.774620, 1.570796, 1.697762],accel_mss,speed_ms,0,blend_radius_m)
    |   movel([0.126917, -1.327918, -2.609712, -0.774759, 1.570796, 1.697714],accel_mss,speed_ms,0,blend_radius_m)
    |   movel([0.126976, -1.327295, -2.610105, -0.774989, 1.570796, 1.697772],accel_mss,speed_ms,0,blend_radius_m)
    |   movel([0.127034, -1.326535, -2.610584, -0.775270, 1.570796, 1.697830],accel_mss,speed_ms,0,blend_radius_m)
    |   movel([0.126915, -1.326132, -2.610837, -0.775419, 1.570796, 1.697712],accel_mss,speed_ms,0,blend_radius_m)
    |   movel([0.126572, -1.325901, -2.610983, -0.775505, 1.570796, 1.697368],accel_mss,speed_ms,0,blend_radius_m)
    |   movel([0.125834, -1.325741, -2.611083, -0.775565, 1.570796, 1.696630],accel_mss,speed_ms,0,blend_radius_m)
    |   movel([0.124274, -1.324872, -2.611629, -0.775888, 1.570796, 1.695070],accel_mss,speed_ms,0,blend_radius_m)
    |   movel([0.123884, -1.323077, -2.612753, -0.776559, 1.570796, 1.694680],accel_mss,speed_ms,0,blend_radius_m)
    |   speed_ms = 0.003
    |   movel([0.123884, -1.326552, -2.614331, -0.771505, 1.570796, 1.694680],accel_mss,speed_ms,0,blend_radius_m)
    |   speed_ms = 0.007
    |   movel([0.124792, -1.324351, -2.615711, -0.772327, 1.570796, 1.695588],accel_mss,speed_ms,0,blend_radius_m)
    |   movel([0.126733, -1.322386, -2.616936, -0.773066, 1.570796, 1.697529],accel_mss,speed_ms,0,blend_radius_m)
    |   movel([0.127638, -1.321695, -2.617366, -0.773328, 1.570796, 1.698435],accel_mss,speed_ms,0,blend_radius_m)
    |   movel([0.128111, -1.321198, -2.617675, -0.773516, 1.570796, 1.698907],accel_mss,speed_ms,0,blend_radius_m)
    |   movel([0.128379, -1.320665, -2.618006, -0.773718, 1.570796, 1.699175],accel_mss,speed_ms,0,blend_radius_m)
    |   movel([0.128550, -1.319879, -2.618493, -0.774017, 1.570796, 1.699347],accel_mss,speed_ms,0,blend_radius_m)
    |   movel([0.128674, -1.319239, -2.618889, -0.774261, 1.570796, 1.699471],accel_mss,speed_ms,0,blend_radius_m)
    |   movel([0.128842, -1.318799, -2.619161, -0.774429, 1.570796, 1.699638],accel_mss,speed_ms,0,blend_radius_m)
    |   movel([0.129067, -1.318514, -2.619337, -0.774538, 1.570796, 1.699864],accel_mss,speed_ms,0,blend_radius_m)
    |   movel([0.129356, -1.318347, -2.619440, -0.774602, 1.570796, 1.700152],accel_mss,speed_ms,0,blend_radius_m)
    |   movel([0.129619, -1.318354, -2.619435, -0.774599, 1.570796, 1.700416],accel_mss,speed_ms,0,blend_radius_m)
    |   movel([0.129777, -1.318533, -2.619325, -0.774531, 1.570796, 1.700573],accel_mss,speed_ms,0,blend_radius_m)
    |   movel([0.129825, -1.318916, -2.619089, -0.774385, 1.570796, 1.700621],accel_mss,speed_ms,0,blend_radius_m)
    |   movel([0.129763, -1.319549, -2.618697, -0.774143, 1.570796, 1.700559],accel_mss,speed_ms,0,blend_radius_m)
    |   movel([0.129702, -1.320320, -2.618220, -0.773849, 1.570796, 1.700498],accel_mss,speed_ms,0,blend_radius_m)
    |   movel([0.129820, -1.320728, -2.617967, -0.773694, 1.570796, 1.700617],accel_mss,speed_ms,0,blend_radius_m)
    |   movel([0.130166, -1.320962, -2.617822, -0.773605, 1.570796, 1.700962],accel_mss,speed_ms,0,blend_radius_m)
    |   movel([0.130909, -1.321123, -2.617721, -0.773544, 1.570796, 1.701705],accel_mss,speed_ms,0,blend_radius_m)
    |   movel([0.131488, -1.321272, -2.617629, -0.773488, 1.570796, 1.702285],accel_mss,speed_ms,0,blend_radius_m)
    |   movel([0.131996, -1.321539, -2.617463, -0.773387, 1.570796, 1.702792],accel_mss,speed_ms,0,blend_radius_m)
    |   movel([0.132396, -1.321900, -2.617239, -0.773250, 1.570796, 1.703192],accel_mss,speed_ms,0,blend_radius_m)
    |   movel([0.132649, -1.322327, -2.616973, -0.773089, 1.570796, 1.703446],accel_mss,speed_ms,0,blend_radius_m)
    |   movel([0.132924, -1.323194, -2.616433, -0.772762, 1.570796, 1.703720],accel_mss,speed_ms,0,blend_radius_m)
    |   movel([0.132947, -1.323825, -2.616040, -0.772525, 1.570796, 1.703744],accel_mss,speed_ms,0,blend_radius_m)
    |   movel([0.132731, -1.324529, -2.615599, -0.772260, 1.570796, 1.703527],accel_mss,speed_ms,0,blend_radius_m)
    |   movel([0.132168, -1.325645, -2.614901, -0.771844, 1.570796, 1.702965],accel_mss,speed_ms,0,blend_radius_m)
    |   movel([0.131743, -1.326309, -2.614484, -0.771596, 1.570796, 1.702540],accel_mss,speed_ms,0,blend_radius_m)
    |   movel([0.131210, -1.326946, -2.614084, -0.771359, 1.570796, 1.702006],accel_mss,speed_ms,0,blend_radius_m)
    |   movel([0.130584, -1.327533, -2.613715, -0.771141, 1.570796, 1.701380],accel_mss,speed_ms,0,blend_radius_m)
    |   movel([0.129887, -1.328054, -2.613386, -0.770948, 1.570796, 1.700683],accel_mss,speed_ms,0,blend_radius_m)
    |   movel([0.129036, -1.328667, -2.613000, -0.770722, 1.570796, 1.699832],accel_mss,speed_ms,0,blend_radius_m)
    |   movel([0.128593, -1.329122, -2.612713, -0.770554, 1.570796, 1.699389],accel_mss,speed_ms,0,blend_radius_m)
    |   movel([0.128342, -1.329629, -2.612392, -0.770367, 1.570796, 1.699139],accel_mss,speed_ms,0,blend_radius_m)
    |   movel([0.128176, -1.330419, -2.611893, -0.770078, 1.570796, 1.698973],accel_mss,speed_ms,0,blend_radius_m)
    |   movel([0.128053, -1.331059, -2.611487, -0.769843, 1.570796, 1.698849],accel_mss,speed_ms,0,blend_radius_m)
    |   movel([0.127887, -1.331495, -2.611210, -0.769684, 1.570796, 1.698683],accel_mss,speed_ms,0,blend_radius_m)
    |   movel([0.127665, -1.331778, -2.611030, -0.769580, 1.570796, 1.698461],accel_mss,speed_ms,0,blend_radius_m)
    |   movel([0.127381, -1.331940, -2.610928, -0.769521, 1.570796, 1.698177],accel_mss,speed_ms,0,blend_radius_m)
    |   movel([0.127121, -1.331932, -2.610932, -0.769524, 1.570796, 1.697918],accel_mss,speed_ms,0,blend_radius_m)
    |   movel([0.126965, -1.331757, -2.611044, -0.769588, 1.570796, 1.697762],accel_mss,speed_ms,0,blend_radius_m)
    |   movel([0.126917, -1.331381, -2.611282, -0.769725, 1.570796, 1.697714],accel_mss,speed_ms,0,blend_radius_m)
    |   movel([0.126976, -1.330760, -2.611676, -0.769953, 1.570796, 1.697772],accel_mss,speed_ms,0,blend_radius_m)
    |   movel([0.127034, -1.330002, -2.612157, -0.770231, 1.570796, 1.697830],accel_mss,speed_ms,0,blend_radius_m)
    |   movel([0.126915, -1.329600, -2.612411, -0.770378, 1.570796, 1.697712],accel_mss,speed_ms,0,blend_radius_m)
    |   movel([0.126572, -1.329369, -2.612557, -0.770463, 1.570796, 1.697368],accel_mss,speed_ms,0,blend_radius_m)
    |   movel([0.125834, -1.329210, -2.612657, -0.770522, 1.570796, 1.696630],accel_mss,speed_ms,0,blend_radius_m)
    |   movel([0.124274, -1.328343, -2.613205, -0.770842, 1.570796, 1.695070],accel_mss,speed_ms,0,blend_radius_m)
    |   movel([0.123884, -1.326552, -2.614331, -0.771505, 1.570796, 1.694680],accel_mss,speed_ms,0,blend_radius_m)
    |   speed_ms = 0.003
    |   # Splitting Linear movement in 8 (instruction 491: MoveL 457)
    |   movel([0.123884, -1.324811, -2.613543, -0.774035, 1.570796, 1.694680],accel_mss,speed_ms,0,blend_radius_m)
    |   movel([0.123884, -1.323077, -2.612753, -0.776559, 1.570796, 1.694680],accel_mss,speed_ms,0,blend_radius_m)
    |   movel([0.123884, -1.321350, -2.611960, -0.779079, 1.570796, 1.694680],accel_mss,speed_ms,0,blend_radius_m)
    |   movel([0.123884, -1.319629, -2.611165, -0.781595, 1.570796, 1.694680],accel_mss,speed_ms,0,blend_radius_m)
    |   movel([0.123884, -1.317914, -2.610369, -0.784106, 1.570796, 1.694680],accel_mss,speed_ms,0,blend_radius_m)
    |   movel([0.123884, -1.316206, -2.609570, -0.786613, 1.570796, 1.694680],accel_mss,speed_ms,0,blend_radius_m)
    |   movel([0.123884, -1.314505, -2.608769, -0.789115, 1.570796, 1.694680],accel_mss,speed_ms,0,blend_radius_m)
    |   movel([0.123884, -1.312811, -2.607966, -0.791612, 1.570796, 1.694680],accel_mss,speed_ms,0,blend_radius_m)
    |   speed_ms = 1.000
    |   # Splitting Linear movement in 12 (instruction 493: MoveL 458)
    |   movel([0.123884, -1.310561, -2.606892, -0.794936, 1.570796, 1.694680],accel_mss,speed_ms,0,blend_radius_m)
    |   movel([0.123884, -1.308324, -2.605815, -0.798251, 1.570796, 1.694680],accel_mss,speed_ms,0,blend_radius_m)
    |   movel([0.123884, -1.306098, -2.604734, -0.801558, 1.570796, 1.694680],accel_mss,speed_ms,0,blend_radius_m)
    |   movel([0.123884, -1.303883, -2.603649, -0.804857, 1.570796, 1.694680],accel_mss,speed_ms,0,blend_radius_m)
    |   movel([0.123884, -1.301681, -2.602560, -0.808148, 1.570796, 1.694680],accel_mss,speed_ms,0,blend_radius_m)
    |   movel([0.123884, -1.299489, -2.601468, -0.811431, 1.570796, 1.694680],accel_mss,speed_ms,0,blend_radius_m)
    |   movel([0.123884, -1.297310, -2.600373, -0.814706, 1.570796, 1.694680],accel_mss,speed_ms,0,blend_radius_m)
    |   movel([0.123884, -1.295142, -2.599274, -0.817973, 1.570796, 1.694680],accel_mss,speed_ms,0,blend_radius_m)
    |   movel([0.123884, -1.292985, -2.598171, -0.821233, 1.570796, 1.694680],accel_mss,speed_ms,0,blend_radius_m)
    |   movel([0.123884, -1.290840, -2.597065, -0.824484, 1.570796, 1.694680],accel_mss,speed_ms,0,blend_radius_m)
    |   movel([0.123884, -1.288706, -2.595956, -0.827727, 1.570796, 1.694680],accel_mss,speed_ms,0,blend_radius_m)
    |   movel([0.123884, -1.286584, -2.594843, -0.830963, 1.570796, 1.694680],accel_mss,speed_ms,0,blend_radius_m)
    |   # Splitting Linear movement in 6 (instruction 494: MoveL 459)
    |   movel([0.126335, -1.285873, -2.595264, -0.831252, 1.570796, 1.697132],accel_mss,speed_ms,0,blend_radius_m)
    |   movel([0.128788, -1.285166, -2.595682, -0.831541, 1.570796, 1.699585],accel_mss,speed_ms,0,blend_radius_m)
    |   movel([0.131242, -1.284463, -2.596097, -0.831828, 1.570796, 1.702039],accel_mss,speed_ms,0,blend_radius_m)
    |   movel([0.133698, -1.283765, -2.596509, -0.832115, 1.570796, 1.704494],accel_mss,speed_ms,0,blend_radius_m)
    |   movel([0.136154, -1.283070, -2.596918, -0.832401, 1.570796, 1.706950],accel_mss,speed_ms,0,blend_radius_m)
    |   movel([0.138612, -1.282379, -2.597325, -0.832685, 1.570796, 1.709408],accel_mss,speed_ms,0,blend_radius_m)
    |   # Splitting Linear movement in 14 (instruction 495: MoveL 460)
    |   movel([0.138612, -1.284202, -2.598283, -0.829904, 1.570796, 1.709408],accel_mss,speed_ms,0,blend_radius_m)
    |   movel([0.138612, -1.286033, -2.599238, -0.827118, 1.570796, 1.709408],accel_mss,speed_ms,0,blend_radius_m)
    |   movel([0.138612, -1.287872, -2.600191, -0.824325, 1.570796, 1.709408],accel_mss,speed_ms,0,blend_radius_m)
    |   movel([0.138612, -1.289720, -2.601142, -0.821527, 1.570796, 1.709408],accel_mss,speed_ms,0,blend_radius_m)
    |   movel([0.138612, -1.291577, -2.602090, -0.818722, 1.570796, 1.709408],accel_mss,speed_ms,0,blend_radius_m)
    |   movel([0.138612, -1.293442, -2.603035, -0.815912, 1.570796, 1.709408],accel_mss,speed_ms,0,blend_radius_m)
    |   movel([0.138612, -1.295315, -2.603978, -0.813096, 1.570796, 1.709408],accel_mss,speed_ms,0,blend_radius_m)
    |   movel([0.138612, -1.297197, -2.604918, -0.810274, 1.570796, 1.709408],accel_mss,speed_ms,0,blend_radius_m)
    |   movel([0.138612, -1.299088, -2.605855, -0.807446, 1.570796, 1.709408],accel_mss,speed_ms,0,blend_radius_m)
    |   movel([0.138612, -1.300987, -2.606790, -0.804612, 1.570796, 1.709408],accel_mss,speed_ms,0,blend_radius_m)
    |   movel([0.138612, -1.302895, -2.607722, -0.801771, 1.570796, 1.709408],accel_mss,speed_ms,0,blend_radius_m)
    |   movel([0.138612, -1.304812, -2.608652, -0.798925, 1.570796, 1.709408],accel_mss,speed_ms,0,blend_radius_m)
    |   movel([0.138612, -1.306737, -2.609579, -0.796073, 1.570796, 1.709408],accel_mss,speed_ms,0,blend_radius_m)
    |   movel([0.138612, -1.308670, -2.610503, -0.793216, 1.570796, 1.709408],accel_mss,speed_ms,0,blend_radius_m)
    |   speed_ms = 0.003
    |   # Splitting Linear movement in 6 (instruction 497: MoveL 461)
    |   movel([0.138612, -1.310370, -2.611309, -0.790710, 1.570796, 1.709408],accel_mss,speed_ms,0,blend_radius_m)
    |   movel([0.138612, -1.312076, -2.612114, -0.788200, 1.570796, 1.709408],accel_mss,speed_ms,0,blend_radius_m)
    |   movel([0.138612, -1.313788, -2.612916, -0.785685, 1.570796, 1.709408],accel_mss,speed_ms,0,blend_radius_m)
    |   movel([0.138612, -1.315507, -2.613716, -0.783165, 1.570796, 1.709408],accel_mss,speed_ms,0,blend_radius_m)
    |   movel([0.138612, -1.317233, -2.614514, -0.780642, 1.570796, 1.709408],accel_mss,speed_ms,0,blend_radius_m)
    |   movel([0.138612, -1.318966, -2.615310, -0.778113, 1.570796, 1.709408],accel_mss,speed_ms,0,blend_radius_m)
    |   speed_ms = 0.007
    |   movel([0.138808, -1.318037, -2.615885, -0.778467, 1.570796, 1.709604],accel_mss,speed_ms,0,blend_radius_m)
    |   movel([0.139084, -1.317339, -2.616316, -0.778734, 1.570796, 1.709880],accel_mss,speed_ms,0,blend_radius_m)
    |   movel([0.139519, -1.316683, -2.616721, -0.778985, 1.570796, 1.710315],accel_mss,speed_ms,0,blend_radius_m)
    |   movel([0.140221, -1.315890, -2.617209, -0.779290, 1.570796, 1.711018],accel_mss,speed_ms,0,blend_radius_m)
    |   movel([0.140787, -1.315344, -2.617545, -0.779500, 1.570796, 1.711584],accel_mss,speed_ms,0,blend_radius_m)
    |   movel([0.141366, -1.314853, -2.617846, -0.779689, 1.570796, 1.712162],accel_mss,speed_ms,0,blend_radius_m)
    |   movel([0.141880, -1.314475, -2.618078, -0.779835, 1.570796, 1.712677],accel_mss,speed_ms,0,blend_radius_m)
    |   movel([0.142213, -1.314317, -2.618175, -0.779897, 1.570796, 1.713009],accel_mss,speed_ms,0,blend_radius_m)
    |   movel([0.142531, -1.314136, -2.618286, -0.779967, 1.570796, 1.713327],accel_mss,speed_ms,0,blend_radius_m)
    |   movel([0.142772, -1.313825, -2.618477, -0.780087, 1.570796, 1.713568],accel_mss,speed_ms,0,blend_radius_m)
    |   movel([0.142956, -1.313320, -2.618786, -0.780283, 1.570796, 1.713752],accel_mss,speed_ms,0,blend_radius_m)
    |   movel([0.143116, -1.312497, -2.619289, -0.780603, 1.570796, 1.713913],accel_mss,speed_ms,0,blend_radius_m)
    |   movel([0.143274, -1.311694, -2.619779, -0.780916, 1.570796, 1.714070],accel_mss,speed_ms,0,blend_radius_m)
    |   movel([0.143457, -1.311179, -2.620093, -0.781117, 1.570796, 1.714254],accel_mss,speed_ms,0,blend_radius_m)
    |   movel([0.143690, -1.310859, -2.620288, -0.781242, 1.570796, 1.714486],accel_mss,speed_ms,0,blend_radius_m)
    |   movel([0.143991, -1.310679, -2.620397, -0.781312, 1.570796, 1.714787],accel_mss,speed_ms,0,blend_radius_m)
    |   movel([0.144256, -1.310694, -2.620388, -0.781307, 1.570796, 1.715052],accel_mss,speed_ms,0,blend_radius_m)
    |   movel([0.144406, -1.310885, -2.620272, -0.781232, 1.570796, 1.715202],accel_mss,speed_ms,0,blend_radius_m)
    |   movel([0.144446, -1.311294, -2.620023, -0.781072, 1.570796, 1.715243],accel_mss,speed_ms,0,blend_radius_m)
    |   movel([0.144364, -1.311978, -2.619606, -0.780805, 1.570796, 1.715160],accel_mss,speed_ms,0,blend_radius_m)
    |   movel([0.144277, -1.312805, -2.619101, -0.780483, 1.570796, 1.715073],accel_mss,speed_ms,0,blend_radius_m)
    |   movel([0.144375, -1.313236, -2.618837, -0.780316, 1.570796, 1.715172],accel_mss,speed_ms,0,blend_radius_m)
    |   movel([0.144697, -1.313483, -2.618686, -0.780220, 1.570796, 1.715493],accel_mss,speed_ms,0,blend_radius_m)
    |   movel([0.145385, -1.313650, -2.618584, -0.780155, 1.570796, 1.716182],accel_mss,speed_ms,0,blend_radius_m)
    |   movel([0.145903, -1.313786, -2.618501, -0.780102, 1.570796, 1.716699],accel_mss,speed_ms,0,blend_radius_m)
    |   movel([0.146421, -1.314026, -2.618354, -0.780009, 1.570796, 1.717217],accel_mss,speed_ms,0,blend_radius_m)
    |   movel([0.146865, -1.314324, -2.618171, -0.779894, 1.570796, 1.717661],accel_mss,speed_ms,0,blend_radius_m)
    |   movel([0.147148, -1.314638, -2.617979, -0.779773, 1.570796, 1.717945],accel_mss,speed_ms,0,blend_radius_m)
    |   movel([0.147487, -1.316003, -2.617140, -0.779246, 1.570796, 1.718284],accel_mss,speed_ms,0,blend_radius_m)
    |   movel([0.147058, -1.317700, -2.616093, -0.778596, 1.570796, 1.717855],accel_mss,speed_ms,0,blend_radius_m)
    |   movel([0.145965, -1.319370, -2.615060, -0.777959, 1.570796, 1.716762],accel_mss,speed_ms,0,blend_radius_m)
    |   movel([0.144430, -1.320660, -2.614259, -0.777470, 1.570796, 1.715226],accel_mss,speed_ms,0,blend_radius_m)
    |   movel([0.143768, -1.321120, -2.613973, -0.777296, 1.570796, 1.714565],accel_mss,speed_ms,0,blend_radius_m)
    |   movel([0.143394, -1.321533, -2.613716, -0.777140, 1.570796, 1.714191],accel_mss,speed_ms,0,blend_radius_m)
    |   movel([0.143164, -1.322060, -2.613388, -0.776942, 1.570796, 1.713960],accel_mss,speed_ms,0,blend_radius_m)
    |   movel([0.142980, -1.322965, -2.612822, -0.776601, 1.570796, 1.713776],accel_mss,speed_ms,0,blend_radius_m)
    |   movel([0.142812, -1.323836, -2.612278, -0.776275, 1.570796, 1.713608],accel_mss,speed_ms,0,blend_radius_m)
    |   movel([0.142626, -1.324291, -2.611993, -0.776105, 1.570796, 1.713423],accel_mss,speed_ms,0,blend_radius_m)
    |   movel([0.142352, -1.324567, -2.611820, -0.776002, 1.570796, 1.713149],accel_mss,speed_ms,0,blend_radius_m)
    |   movel([0.141926, -1.324757, -2.611701, -0.775931, 1.570796, 1.712723],accel_mss,speed_ms,0,blend_radius_m)
    |   movel([0.141525, -1.324794, -2.611678, -0.775917, 1.570796, 1.712321],accel_mss,speed_ms,0,blend_radius_m)
    |   movel([0.141316, -1.324646, -2.611771, -0.775972, 1.570796, 1.712112],accel_mss,speed_ms,0,blend_radius_m)
    |   movel([0.141267, -1.324246, -2.612021, -0.776122, 1.570796, 1.712063],accel_mss,speed_ms,0,blend_radius_m)
    |   movel([0.141382, -1.323363, -2.612574, -0.776452, 1.570796, 1.712178],accel_mss,speed_ms,0,blend_radius_m)
    |   movel([0.141480, -1.322569, -2.613070, -0.776750, 1.570796, 1.712276],accel_mss,speed_ms,0,blend_radius_m)
    |   movel([0.141447, -1.322130, -2.613343, -0.776915, 1.570796, 1.712244],accel_mss,speed_ms,0,blend_radius_m)
    |   movel([0.141289, -1.321933, -2.613466, -0.776989, 1.570796, 1.712085],accel_mss,speed_ms,0,blend_radius_m)
    |   movel([0.141004, -1.321920, -2.613475, -0.776994, 1.570796, 1.711801],accel_mss,speed_ms,0,blend_radius_m)
    |   movel([0.140696, -1.321941, -2.613461, -0.776986, 1.570796, 1.711492],accel_mss,speed_ms,0,blend_radius_m)
    |   movel([0.140263, -1.321829, -2.613531, -0.777028, 1.570796, 1.711059],accel_mss,speed_ms,0,blend_radius_m)
    |   movel([0.139796, -1.321633, -2.613654, -0.777102, 1.570796, 1.710593],accel_mss,speed_ms,0,blend_radius_m)
    |   movel([0.139361, -1.321371, -2.613817, -0.777201, 1.570796, 1.710157],accel_mss,speed_ms,0,blend_radius_m)
    |   movel([0.138857, -1.320919, -2.614098, -0.777372, 1.570796, 1.709653],accel_mss,speed_ms,0,blend_radius_m)
    |   movel([0.138597, -1.320461, -2.614383, -0.777545, 1.570796, 1.709393],accel_mss,speed_ms,0,blend_radius_m)
    |   movel([0.138523, -1.319863, -2.614754, -0.777772, 1.570796, 1.709320],accel_mss,speed_ms,0,blend_radius_m)
    |   movel([0.138612, -1.318966, -2.615310, -0.778113, 1.570796, 1.709408],accel_mss,speed_ms,0,blend_radius_m)
    |   speed_ms = 0.003
    |   movel([0.138612, -1.322451, -2.616896, -0.773042, 1.570796, 1.709408],accel_mss,speed_ms,0,blend_radius_m)
    |   speed_ms = 0.007
    |   movel([0.138808, -1.321525, -2.617472, -0.773392, 1.570796, 1.709604],accel_mss,speed_ms,0,blend_radius_m)
    |   movel([0.139084, -1.320828, -2.617905, -0.773656, 1.570796, 1.709880],accel_mss,speed_ms,0,blend_radius_m)
    |   movel([0.139519, -1.320174, -2.618310, -0.773905, 1.570796, 1.710315],accel_mss,speed_ms,0,blend_radius_m)
    |   movel([0.140221, -1.319382, -2.618800, -0.774206, 1.570796, 1.711018],accel_mss,speed_ms,0,blend_radius_m)
    |   movel([0.140787, -1.318838, -2.619136, -0.774414, 1.570796, 1.711584],accel_mss,speed_ms,0,blend_radius_m)
    |   movel([0.141366, -1.318349, -2.619439, -0.774602, 1.570796, 1.712162],accel_mss,speed_ms,0,blend_radius_m)
    |   movel([0.141880, -1.317971, -2.619671, -0.774746, 1.570796, 1.712677],accel_mss,speed_ms,0,blend_radius_m)
    |   movel([0.142213, -1.317814, -2.619769, -0.774806, 1.570796, 1.713009],accel_mss,speed_ms,0,blend_radius_m)
    |   movel([0.142531, -1.317633, -2.619880, -0.774876, 1.570796, 1.713327],accel_mss,speed_ms,0,blend_radius_m)
    |   movel([0.142772, -1.317322, -2.620071, -0.774995, 1.570796, 1.713568],accel_mss,speed_ms,0,blend_radius_m)
    |   movel([0.142956, -1.316819, -2.620381, -0.775189, 1.570796, 1.713752],accel_mss,speed_ms,0,blend_radius_m)
    |   movel([0.143116, -1.315997, -2.620886, -0.775506, 1.570796, 1.713913],accel_mss,speed_ms,0,blend_radius_m)
    |   movel([0.143274, -1.315196, -2.621377, -0.775815, 1.570796, 1.714070],accel_mss,speed_ms,0,blend_radius_m)
    |   movel([0.143457, -1.314683, -2.621692, -0.776014, 1.570796, 1.714254],accel_mss,speed_ms,0,blend_radius_m)
    |   movel([0.143690, -1.314364, -2.621887, -0.776138, 1.570796, 1.714486],accel_mss,speed_ms,0,blend_radius_m)
    |   movel([0.143991, -1.314184, -2.621997, -0.776208, 1.570796, 1.714787],accel_mss,speed_ms,0,blend_radius_m)
    |   movel([0.144256, -1.314199, -2.621988, -0.776202, 1.570796, 1.715052],accel_mss,speed_ms,0,blend_radius_m)
    |   movel([0.144406, -1.314390, -2.621871, -0.776128, 1.570796, 1.715202],accel_mss,speed_ms,0,blend_radius_m)
    |   movel([0.144446, -1.314797, -2.621622, -0.775970, 1.570796, 1.715243],accel_mss,speed_ms,0,blend_radius_m)
    |   movel([0.144364, -1.315480, -2.621203, -0.775705, 1.570796, 1.715160],accel_mss,speed_ms,0,blend_radius_m)
    |   movel([0.144277, -1.316305, -2.620697, -0.775387, 1.570796, 1.715073],accel_mss,speed_ms,0,blend_radius_m)
    |   movel([0.144375, -1.316735, -2.620433, -0.775221, 1.570796, 1.715172],accel_mss,speed_ms,0,blend_radius_m)
    |   movel([0.144697, -1.316982, -2.620281, -0.775126, 1.570796, 1.715493],accel_mss,speed_ms,0,blend_radius_m)
    |   movel([0.145385, -1.317148, -2.620179, -0.775062, 1.570796, 1.716182],accel_mss,speed_ms,0,blend_radius_m)
    |   movel([0.145903, -1.317283, -2.620095, -0.775010, 1.570796, 1.716699],accel_mss,speed_ms,0,blend_radius_m)
    |   movel([0.146421, -1.317523, -2.619948, -0.774918, 1.570796, 1.717217],accel_mss,speed_ms,0,blend_radius_m)
    |   movel([0.146865, -1.317820, -2.619765, -0.774804, 1.570796, 1.717661],accel_mss,speed_ms,0,blend_radius_m)
    |   movel([0.147148, -1.318134, -2.619572, -0.774684, 1.570796, 1.717945],accel_mss,speed_ms,0,blend_radius_m)
    |   movel([0.147487, -1.319495, -2.618730, -0.774163, 1.570796, 1.718284],accel_mss,speed_ms,0,blend_radius_m)
    |   movel([0.147058, -1.321189, -2.617681, -0.773520, 1.570796, 1.717855],accel_mss,speed_ms,0,blend_radius_m)
    |   movel([0.145965, -1.322854, -2.616645, -0.772890, 1.570796, 1.716762],accel_mss,speed_ms,0,blend_radius_m)
    |   movel([0.144430, -1.324141, -2.615842, -0.772406, 1.570796, 1.715226],accel_mss,speed_ms,0,blend_radius_m)
    |   movel([0.143768, -1.324600, -2.615555, -0.772234, 1.570796, 1.714565],accel_mss,speed_ms,0,blend_radius_m)
    |   movel([0.143394, -1.325012, -2.615297, -0.772080, 1.570796, 1.714191],accel_mss,speed_ms,0,blend_radius_m)
    |   movel([0.143164, -1.325537, -2.614968, -0.771884, 1.570796, 1.713960],accel_mss,speed_ms,0,blend_radius_m)
    |   movel([0.142980, -1.326441, -2.614401, -0.771547, 1.570796, 1.713776],accel_mss,speed_ms,0,blend_radius_m)
    |   movel([0.142812, -1.327309, -2.613856, -0.771224, 1.570796, 1.713608],accel_mss,speed_ms,0,blend_radius_m)
    |   movel([0.142626, -1.327763, -2.613570, -0.771056, 1.570796, 1.713423],accel_mss,speed_ms,0,blend_radius_m)
    |   movel([0.142352, -1.328039, -2.613396, -0.770954, 1.570796, 1.713149],accel_mss,speed_ms,0,blend_radius_m)
    |   movel([0.141926, -1.328228, -2.613277, -0.770884, 1.570796, 1.712723],accel_mss,speed_ms,0,blend_radius_m)
    |   movel([0.141525, -1.328265, -2.613253, -0.770870, 1.570796, 1.712321],accel_mss,speed_ms,0,blend_radius_m)
    |   movel([0.141316, -1.328117, -2.613347, -0.770925, 1.570796, 1.712112],accel_mss,speed_ms,0,blend_radius_m)
    |   movel([0.141267, -1.327718, -2.613598, -0.771073, 1.570796, 1.712063],accel_mss,speed_ms,0,blend_radius_m)
    |   movel([0.141382, -1.326837, -2.614152, -0.771399, 1.570796, 1.712178],accel_mss,speed_ms,0,blend_radius_m)
    |   movel([0.141480, -1.326045, -2.614650, -0.771694, 1.570796, 1.712276],accel_mss,speed_ms,0,blend_radius_m)
